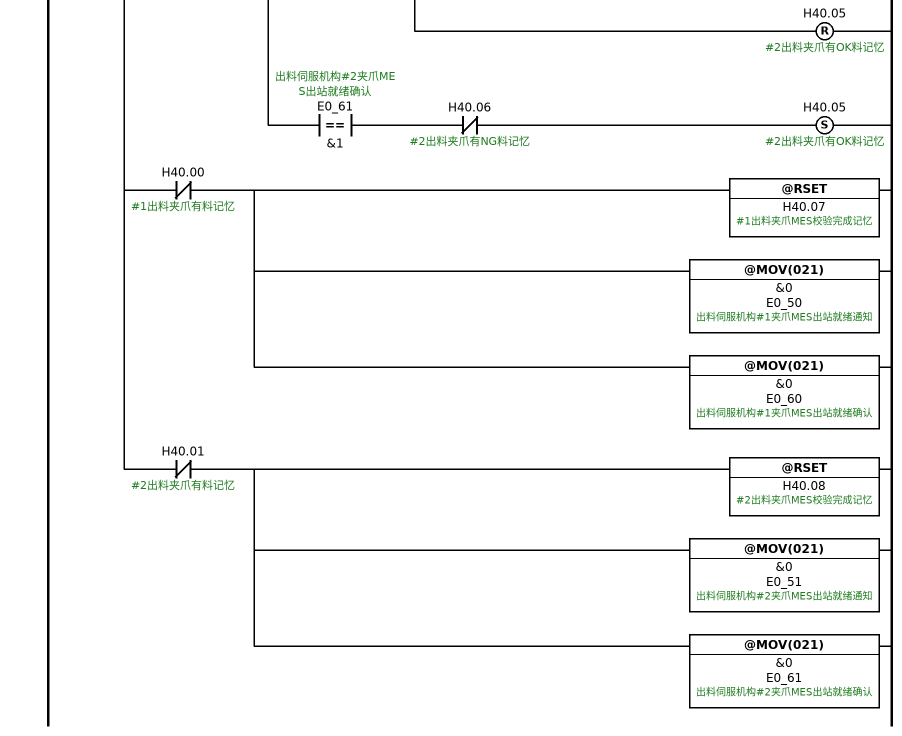
; [picture p408: 出料伺服机构 / Main, rungs 47-47]
; rung 47: 出料伺服机构MES出站校验完成记忆
LD P_On
OUT TR0
AND D1156.05  ; 下料模组夹爪夹紧
OUT TR1
ANDNOT H40.07  ; #1出料夹爪MES校验完成记忆
LD H40.00  ; #1出料夹爪有料记忆
LD>=(325) E0_60 &1  ; 出料伺服机构#1夹爪MES出站就绪确认  // #1出站就绪确认=0：未确认，1：确认OK，
OR H5.07  ; 电脑屏蔽-HMI
OR H5.10  ; 空跑程序
ANDLD
LDNOT H40.00  ; #1出料夹爪有料记忆  // 正常|清尾料时单料状况
AND H40.01  ; #2出料夹爪有料记忆
ORLD
ANDLD
@SET H40.07  ; #1出料夹爪MES校验完成记忆
LD TR1
ANDNOT H40.08  ; #2出料夹爪MES校验完成记忆
LD H40.01  ; #2出料夹爪有料记忆
LD>=(325) E0_61 &1  ; 出料伺服机构#2夹爪MES出站就绪确认  // #2出站就绪确认=0：未确认，1：确认OK，
OR H5.07  ; 电脑屏蔽-HMI
OR H5.10  ; 空跑程序
ANDLD
LDNOT H40.01  ; #2出料夹爪有料记忆  // 正常|清尾料时单料状况
AND H40.00  ; #1出料夹爪有料记忆
ORLD
ANDLD
@SET H40.08  ; #2出料夹爪MES校验完成记忆
LD TR0
AND H40.07  ; #1出料夹爪MES校验完成记忆
LDNOT H6.06  ; MES出站校验使用(1使用)
LD H6.06  ; MES出站校验使用(1使用)
OR P_On
LD H40.03  ; #1出料夹爪有OK料记忆
OR H40.04  ; #1出料夹爪有NG料记忆
ANDLD
ORLD
ANDLD
@MOV(021) &0 E0_50  ; 出料伺服机构#1夹爪MES出站就绪通知
LD TR0
AND H40.08  ; #2出料夹爪MES校验完成记忆
LDNOT H6.06  ; MES出站校验使用(1使用)
LD H6.06  ; MES出站校验使用(1使用)
OR P_On
LD H40.05  ; #2出料夹爪有OK料记忆
OR H40.06  ; #2出料夹爪有NG料记忆
ANDLD
ORLD
ANDLD
@MOV(021) &0 E0_51  ; 出料伺服机构#2夹爪MES出站就绪通知
LD TR0
LD H6.06  ; MES出站校验使用(1使用)
OR P_On
ANDLD
OUT TR1
AND>(320) E0_60 &1  ; 出料伺服机构#1夹爪MES出站就绪确认  // #1出站就绪确认=0：未确认，1：确认OK，
SET H40.04  ; #1出料夹爪有NG料记忆
RSET H40.03  ; #1出料夹爪有OK料记忆
LD TR1
AND=(300) E0_60 &1  ; 出料伺服机构#1夹爪MES出站就绪确认  // #1出站就绪确认=0：未确认，1：确认OK，
ANDNOT H40.04  ; #1出料夹爪有NG料记忆
SET H40.03  ; #1出料夹爪有OK料记忆
LD TR1
AND>(320) E0_61 &1  ; 出料伺服机构#2夹爪MES出站就绪确认  // #1出站就绪确认=0：未确认，1：确认OK，
SET H40.06  ; #2出料夹爪有NG料记忆
RSET H40.05  ; #2出料夹爪有OK料记忆
LD TR1
AND=(300) E0_61 &1  ; 出料伺服机构#2夹爪MES出站就绪确认  // #1出站就绪确认=0：未确认，1：确认OK，
ANDNOT H40.06  ; #2出料夹爪有NG料记忆
SET H40.05  ; #2出料夹爪有OK料记忆
LD TR0
ANDNOT H40.00  ; #1出料夹爪有料记忆
@RSET H40.07  ; #1出料夹爪MES校验完成记忆
@MOV(021) &0 E0_50  ; 出料伺服机构#1夹爪MES出站就绪通知
@MOV(021) &0 E0_60  ; 出料伺服机构#1夹爪MES出站就绪确认
LD TR0
ANDNOT H40.01  ; #2出料夹爪有料记忆
@RSET H40.08  ; #2出料夹爪MES校验完成记忆
@MOV(021) &0 E0_51  ; 出料伺服机构#2夹爪MES出站就绪通知
@MOV(021) &0 E0_61  ; 出料伺服机构#2夹爪MES出站就绪确认

### Section 出料伺服手动

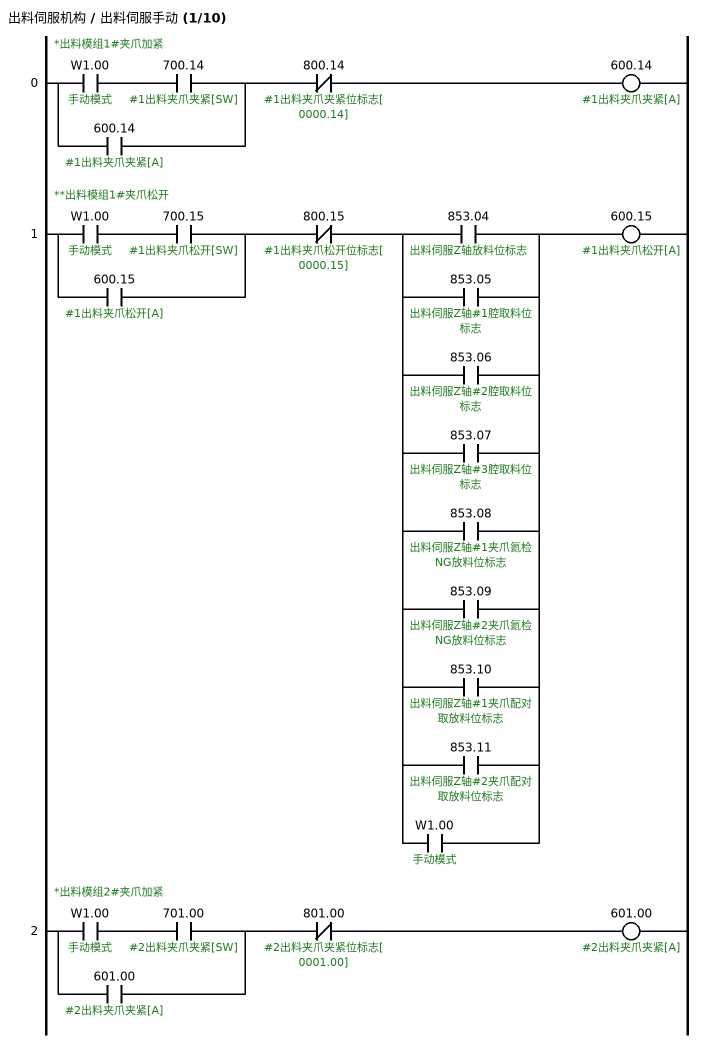
; rung 0: *出料模组1#夹爪加紧
LD W1.00  ; 手动模式
AND 700.14  ; #1出料夹爪夹紧[SW]
OR 600.14  ; #1出料夹爪夹紧[A]
ANDNOT 800.14  ; #1出料夹爪夹紧位标志[0000.14]
OUT 600.14  ; #1出料夹爪夹紧[A]
; rung 1: **出料模组1#夹爪松开
LD W1.00  ; 手动模式
AND 700.15  ; #1出料夹爪松开[SW]
OR 600.15  ; #1出料夹爪松开[A]
ANDNOT 800.15  ; #1出料夹爪松开位标志[0000.15]
LD 853.04  ; 出料伺服Z轴放料位标志
OR 853.05  ; 出料伺服Z轴#1腔取料位标志
OR 853.06  ; 出料伺服Z轴#2腔取料位标志
OR 853.07  ; 出料伺服Z轴#3腔取料位标志
OR 853.08  ; 出料伺服Z轴#1夹爪氦检NG放料位标志
OR 853.09  ; 出料伺服Z轴#2夹爪氦检NG放料位标志
OR 853.10  ; 出料伺服Z轴#1夹爪配对取放料位标志
OR 853.11  ; 出料伺服Z轴#2夹爪配对取放料位标志
OR W1.00  ; 手动模式
ANDLD
OUT 600.15  ; #1出料夹爪松开[A]
; rung 2: *出料模组2#夹爪加紧
LD W1.00  ; 手动模式
AND 701.00  ; #2出料夹爪夹紧[SW]
OR 601.00  ; #2出料夹爪夹紧[A]
ANDNOT 801.00  ; #2出料夹爪夹紧位标志[0001.00]
OUT 601.00  ; #2出料夹爪夹紧[A]

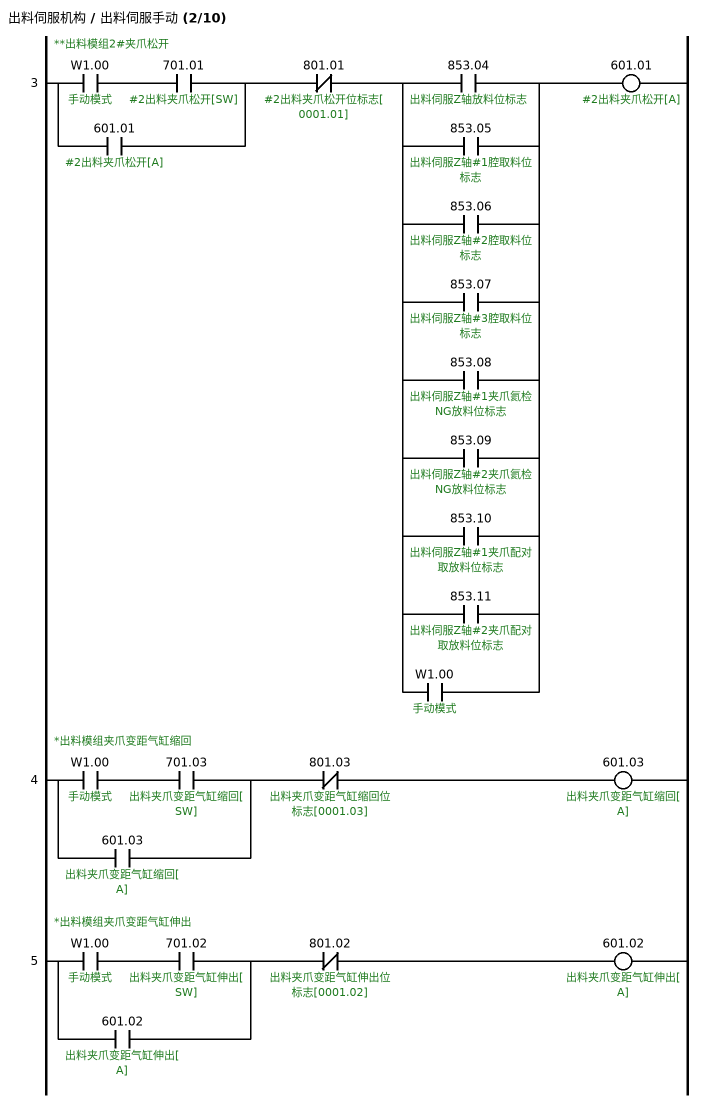
; rung 3: **出料模组2#夹爪松开
LD W1.00  ; 手动模式
AND 701.01  ; #2出料夹爪松开[SW]
OR 601.01  ; #2出料夹爪松开[A]
ANDNOT 801.01  ; #2出料夹爪松开位标志[0001.01]
LD 853.04  ; 出料伺服Z轴放料位标志
OR 853.05  ; 出料伺服Z轴#1腔取料位标志
OR 853.06  ; 出料伺服Z轴#2腔取料位标志
OR 853.07  ; 出料伺服Z轴#3腔取料位标志
OR 853.08  ; 出料伺服Z轴#1夹爪氦检NG放料位标志
OR 853.09  ; 出料伺服Z轴#2夹爪氦检NG放料位标志
OR 853.10  ; 出料伺服Z轴#1夹爪配对取放料位标志
OR 853.11  ; 出料伺服Z轴#2夹爪配对取放料位标志
OR W1.00  ; 手动模式
ANDLD
OUT 601.01  ; #2出料夹爪松开[A]
; rung 4: *出料模组夹爪变距气缸缩回
LD W1.00  ; 手动模式
AND 701.03  ; 出料夹爪变距气缸缩回[SW]
OR 601.03  ; 出料夹爪变距气缸缩回[A]
ANDNOT 801.03  ; 出料夹爪变距气缸缩回位标志[0001.03]
OUT 601.03  ; 出料夹爪变距气缸缩回[A]
; rung 5: *出料模组夹爪变距气缸伸出
LD W1.00  ; 手动模式
AND 701.02  ; 出料夹爪变距气缸伸出[SW]
OR 601.02  ; 出料夹爪变距气缸伸出[A]
ANDNOT 801.02  ; 出料夹爪变距气缸伸出位标志[0001.02]
OUT 601.02  ; 出料夹爪变距气缸伸出[A]

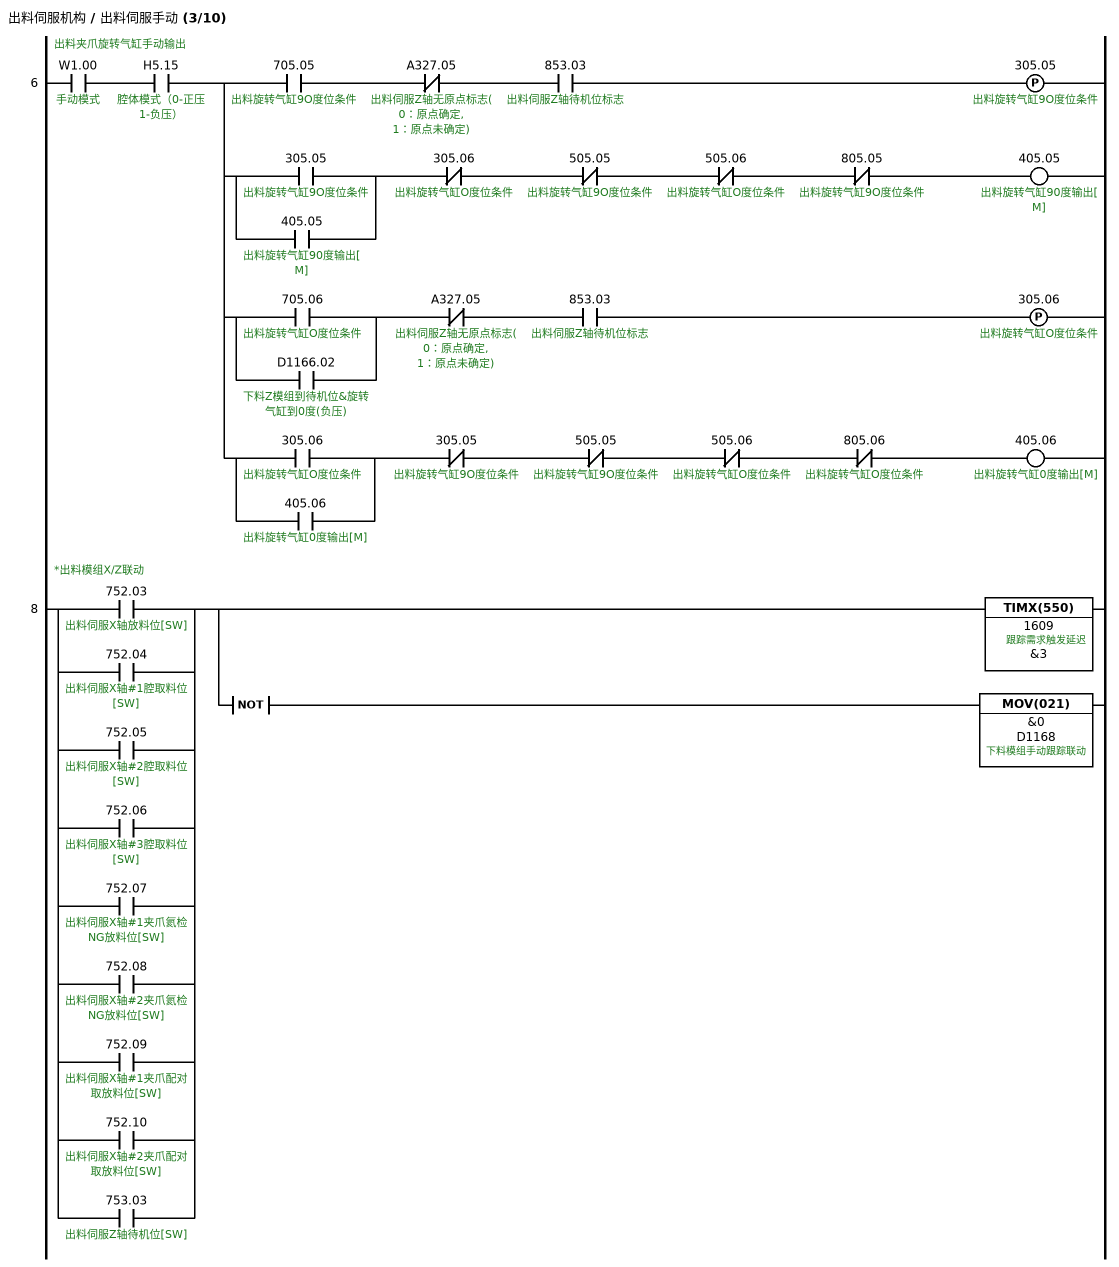
; rung 6: 出料夹爪旋转气缸手动输出
LD W1.00  ; 手动模式
AND H5.15  ; 腔体模式（0-正压 1-负压）
OUT TR0
AND 705.05  ; 出料旋转气缸9O度位条件
ANDNOT A327.05  ; 出料伺服Z轴无原点标志(0：原点确定,1：原点未确定)
AND 853.03  ; 出料伺服Z轴待机位标志
DIFU(013) 305.05  ; 出料旋转气缸9O度位条件
LD TR0
LD 305.05  ; 出料旋转气缸9O度位条件
OR 405.05  ; 出料旋转气缸90度输出[M]
ANDLD
ANDNOT 305.06  ; 出料旋转气缸O度位条件
ANDNOT 505.05  ; 出料旋转气缸9O度位条件
ANDNOT 505.06  ; 出料旋转气缸O度位条件
ANDNOT 805.05  ; 出料旋转气缸9O度位条件
OUT 405.05  ; 出料旋转气缸90度输出[M]
LD TR0
LD 705.06  ; 出料旋转气缸O度位条件
OR D1166.02  ; 下料Z模组到待机位&旋转气缸到0度(负压)
ANDLD
ANDNOT A327.05  ; 出料伺服Z轴无原点标志(0：原点确定,1：原点未确定)
AND 853.03  ; 出料伺服Z轴待机位标志
DIFU(013) 305.06  ; 出料旋转气缸O度位条件
LD TR0
LD 305.06  ; 出料旋转气缸O度位条件
OR 405.06  ; 出料旋转气缸0度输出[M]
ANDLD
ANDNOT 305.05  ; 出料旋转气缸9O度位条件
ANDNOT 505.05  ; 出料旋转气缸9O度位条件
ANDNOT 505.06  ; 出料旋转气缸O度位条件
ANDNOT 805.06  ; 出料旋转气缸O度位条件
OUT 405.06  ; 出料旋转气缸0度输出[M]
; rung 7: ************************** / **************************
; rung 8: *出料模组X/Z联动
LD 752.03  ; 出料伺服X轴放料位[SW]
OR 752.04  ; 出料伺服X轴#1腔取料位[SW]
OR 752.05  ; 出料伺服X轴#2腔取料位[SW]
OR 752.06  ; 出料伺服X轴#3腔取料位[SW]
OR 752.07  ; 出料伺服X轴#1夹爪氦检NG放料位[SW]
OR 752.08  ; 出料伺服X轴#2夹爪氦检NG放料位[SW]
OR 752.09  ; 出料伺服X轴#1夹爪配对取放料位[SW]
OR 752.10  ; 出料伺服X轴#2夹爪配对取放料位[SW]
OR 753.03  ; 出料伺服Z轴待机位[SW]
TIMX(550) 1609 &3  ; 跟踪需求触发延迟
NOT(520)
MOV(021) &0 D1168  ; 下料模组手动跟踪联动

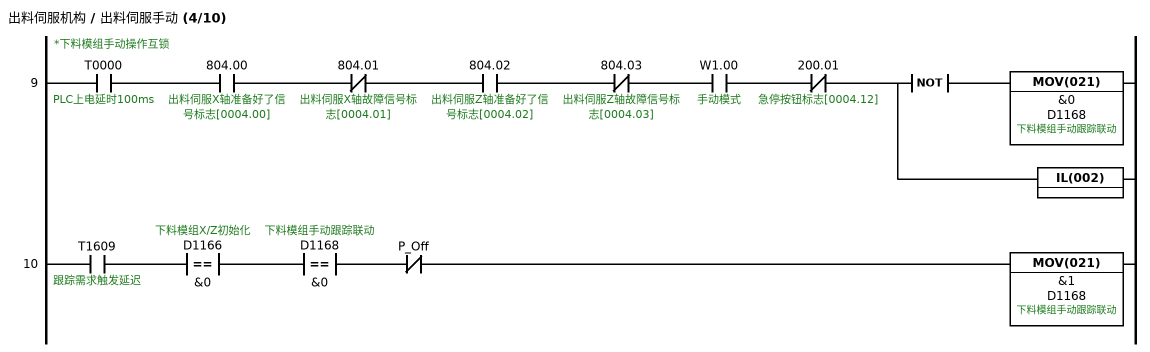
; rung 9: *下料模组手动操作互锁
LD T0000  ; PLC上电延时100ms
AND 804.00  ; 出料伺服X轴准备好了信号标志[0004.00]
ANDNOT 804.01  ; 出料伺服X轴故障信号标志[0004.01]
AND 804.02  ; 出料伺服Z轴准备好了信号标志[0004.02]
ANDNOT 804.03  ; 出料伺服Z轴故障信号标志[0004.03]
AND W1.00  ; 手动模式
ANDNOT 200.01  ; 急停按钮标志[0004.12]
OUT TR0
NOT(520)
MOV(021) &0 D1168  ; 下料模组手动跟踪联动
LD TR0
IL(002)
; rung 10
LD T1609  ; 跟踪需求触发延迟
AND=(300) D1166 &0  ; 下料模组X/Z初始化
AND=(300) D1168 &0  ; 下料模组手动跟踪联动
ANDNOT P_Off
MOV(021) &1 D1168  ; 下料模组手动跟踪联动

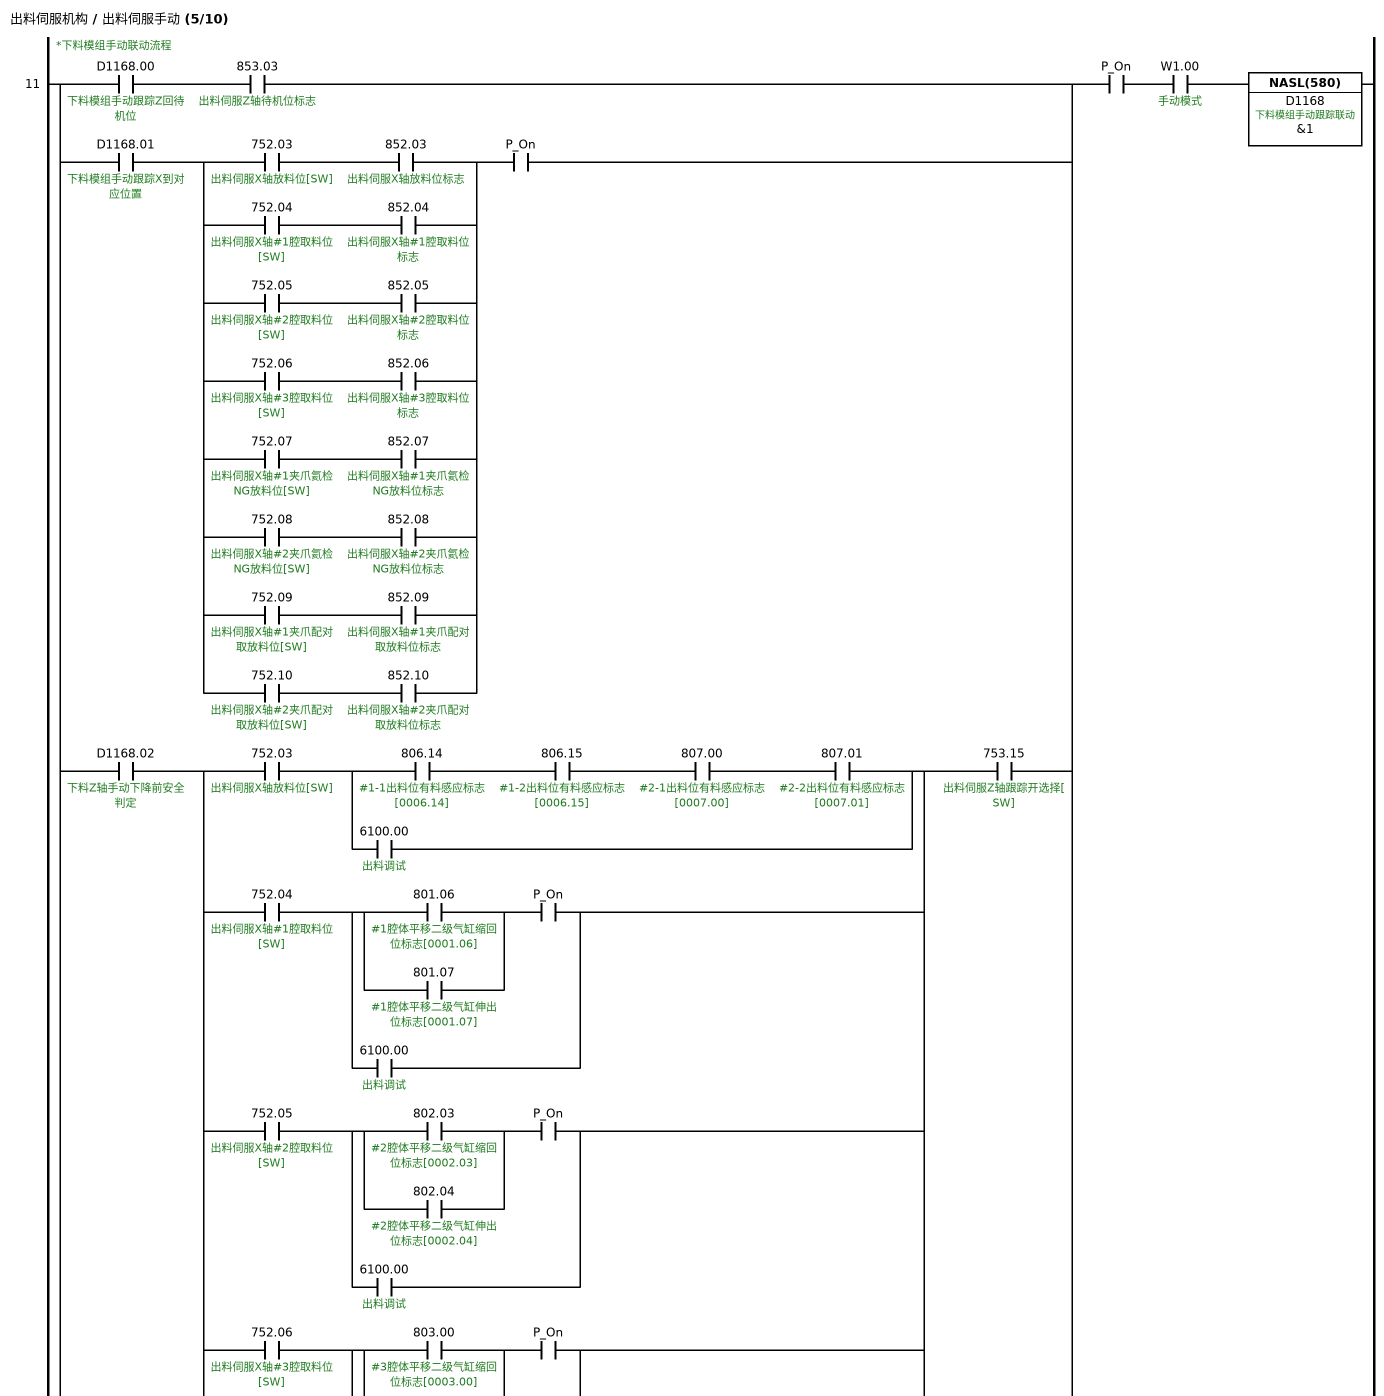

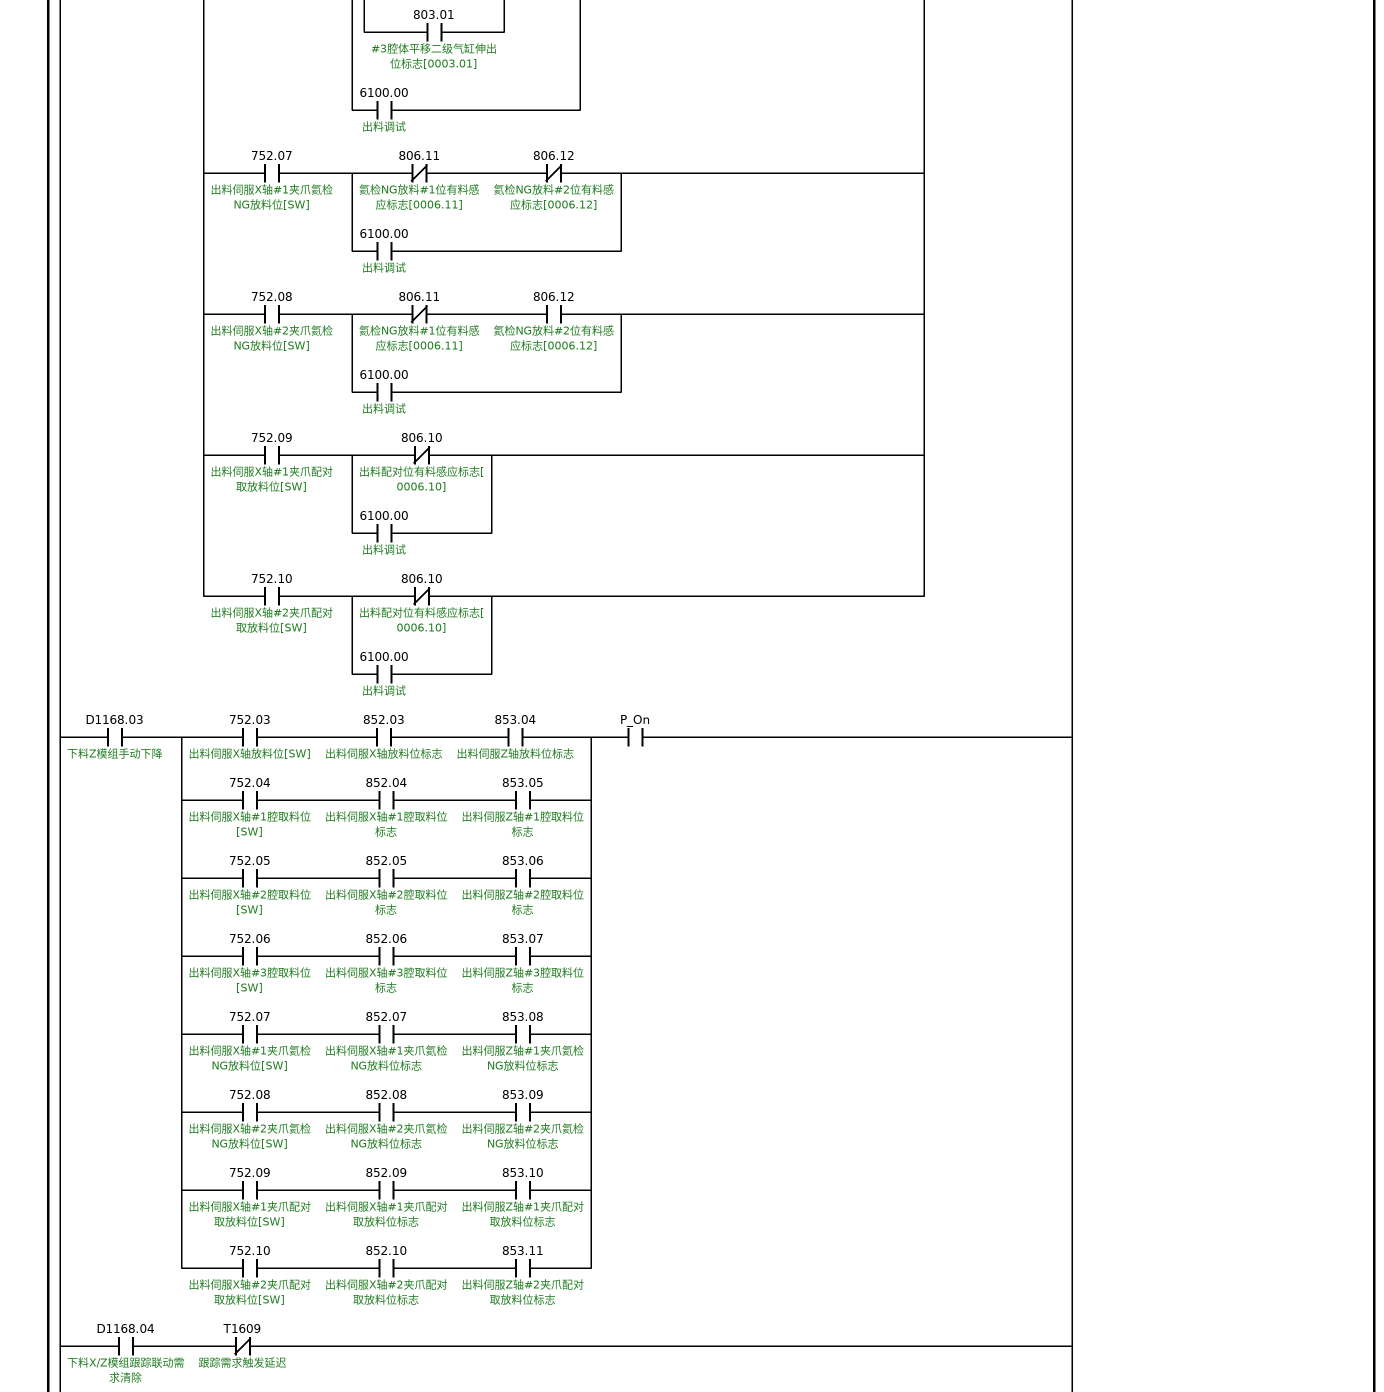

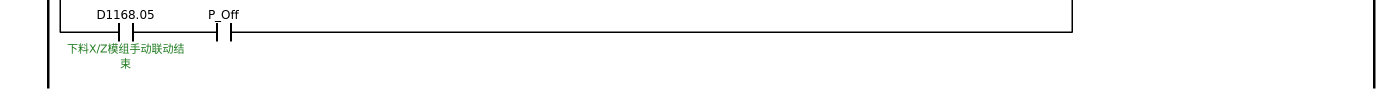
; rung 11: *下料模组手动联动流程
LD D1168.00  ; 下料模组手动跟踪Z回待机位
AND 853.03  ; 出料伺服Z轴待机位标志
LD D1168.01  ; 下料模组手动跟踪X到对应位置
LD 752.03  ; 出料伺服X轴放料位[SW]
AND 852.03  ; 出料伺服X轴放料位标志
LD 752.04  ; 出料伺服X轴#1腔取料位[SW]
AND 852.04  ; 出料伺服X轴#1腔取料位标志
ORLD
LD 752.05  ; 出料伺服X轴#2腔取料位[SW]
AND 852.05  ; 出料伺服X轴#2腔取料位标志
ORLD
LD 752.06  ; 出料伺服X轴#3腔取料位[SW]
AND 852.06  ; 出料伺服X轴#3腔取料位标志
ORLD
LD 752.07  ; 出料伺服X轴#1夹爪氦检NG放料位[SW]
AND 852.07  ; 出料伺服X轴#1夹爪氦检NG放料位标志
ORLD
LD 752.08  ; 出料伺服X轴#2夹爪氦检NG放料位[SW]
AND 852.08  ; 出料伺服X轴#2夹爪氦检NG放料位标志
ORLD
LD 752.09  ; 出料伺服X轴#1夹爪配对取放料位[SW]
AND 852.09  ; 出料伺服X轴#1夹爪配对取放料位标志
ORLD
LD 752.10  ; 出料伺服X轴#2夹爪配对取放料位[SW]
AND 852.10  ; 出料伺服X轴#2夹爪配对取放料位标志
ORLD
ANDLD
AND P_On
ORLD
LD D1168.02  ; 下料Z轴手动下降前安全判定
LD 752.03  ; 出料伺服X轴放料位[SW]
LD 806.14  ; #1-1出料位有料感应标志[0006.14]
AND 806.15  ; #1-2出料位有料感应标志[0006.15]
AND 807.00  ; #2-1出料位有料感应标志[0007.00]
AND 807.01  ; #2-2出料位有料感应标志[0007.01]
OR 6100.00  ; 出料调试
ANDLD
LD 752.04  ; 出料伺服X轴#1腔取料位[SW]
LD 801.06  ; #1腔体平移二级气缸缩回位标志[0001.06]
OR 801.07  ; #1腔体平移二级气缸伸出位标志[0001.07]
AND P_On
OR 6100.00  ; 出料调试
ANDLD
ORLD
LD 752.05  ; 出料伺服X轴#2腔取料位[SW]
LD 802.03  ; #2腔体平移二级气缸缩回位标志[0002.03]
OR 802.04  ; #2腔体平移二级气缸伸出位标志[0002.04]
AND P_On
OR 6100.00  ; 出料调试
ANDLD
ORLD
LD 752.06  ; 出料伺服X轴#3腔取料位[SW]
LD 803.00  ; #3腔体平移二级气缸缩回位标志[0003.00]
OR 803.01  ; #3腔体平移二级气缸伸出位标志[0003.01]
AND P_On
OR 6100.00  ; 出料调试
ANDLD
ORLD
LD 752.07  ; 出料伺服X轴#1夹爪氦检NG放料位[SW]
LDNOT 806.11  ; 氦检NG放料#1位有料感应标志[0006.11]
ANDNOT 806.12  ; 氦检NG放料#2位有料感应标志[0006.12]
OR 6100.00  ; 出料调试
ANDLD
ORLD
LD 752.08  ; 出料伺服X轴#2夹爪氦检NG放料位[SW]
LDNOT 806.11  ; 氦检NG放料#1位有料感应标志[0006.11]
AND 806.12  ; 氦检NG放料#2位有料感应标志[0006.12]
OR 6100.00  ; 出料调试
ANDLD
ORLD
LD 752.09  ; 出料伺服X轴#1夹爪配对取放料位[SW]
LDNOT 806.10  ; 出料配对位有料感应标志[0006.10]
OR 6100.00  ; 出料调试
ANDLD
ORLD
LD 752.10  ; 出料伺服X轴#2夹爪配对取放料位[SW]
LDNOT 806.10  ; 出料配对位有料感应标志[0006.10]
OR 6100.00  ; 出料调试
ANDLD
ORLD
ANDLD
AND 753.15  ; 出料伺服Z轴跟踪开选择[SW]
ORLD
LD D1168.03  ; 下料Z模组手动下降
LD 752.03  ; 出料伺服X轴放料位[SW]
AND 852.03  ; 出料伺服X轴放料位标志
AND 853.04  ; 出料伺服Z轴放料位标志
LD 752.04  ; 出料伺服X轴#1腔取料位[SW]
AND 852.04  ; 出料伺服X轴#1腔取料位标志
AND 853.05  ; 出料伺服Z轴#1腔取料位标志
ORLD
LD 752.05  ; 出料伺服X轴#2腔取料位[SW]
AND 852.05  ; 出料伺服X轴#2腔取料位标志
AND 853.06  ; 出料伺服Z轴#2腔取料位标志
ORLD
LD 752.06  ; 出料伺服X轴#3腔取料位[SW]
AND 852.06  ; 出料伺服X轴#3腔取料位标志
AND 853.07  ; 出料伺服Z轴#3腔取料位标志
ORLD
LD 752.07  ; 出料伺服X轴#1夹爪氦检NG放料位[SW]
AND 852.07  ; 出料伺服X轴#1夹爪氦检NG放料位标志
AND 853.08  ; 出料伺服Z轴#1夹爪氦检NG放料位标志
ORLD
LD 752.08  ; 出料伺服X轴#2夹爪氦检NG放料位[SW]
AND 852.08  ; 出料伺服X轴#2夹爪氦检NG放料位标志
AND 853.09  ; 出料伺服Z轴#2夹爪氦检NG放料位标志
ORLD
LD 752.09  ; 出料伺服X轴#1夹爪配对取放料位[SW]
AND 852.09  ; 出料伺服X轴#1夹爪配对取放料位标志
AND 853.10  ; 出料伺服Z轴#1夹爪配对取放料位标志
ORLD
LD 752.10  ; 出料伺服X轴#2夹爪配对取放料位[SW]
AND 852.10  ; 出料伺服X轴#2夹爪配对取放料位标志
AND 853.11  ; 出料伺服Z轴#2夹爪配对取放料位标志
ORLD
ANDLD
AND P_On
ORLD
LD D1168.04  ; 下料X/Z模组跟踪联动需求清除
ANDNOT T1609  ; 跟踪需求触发延迟
ORLD
LD D1168.05  ; 下料X/Z模组手动联动结束
AND P_Off
ORLD
AND P_On
AND W1.00  ; 手动模式
NASL(580) D1168 &1  ; 下料模组手动跟踪联动

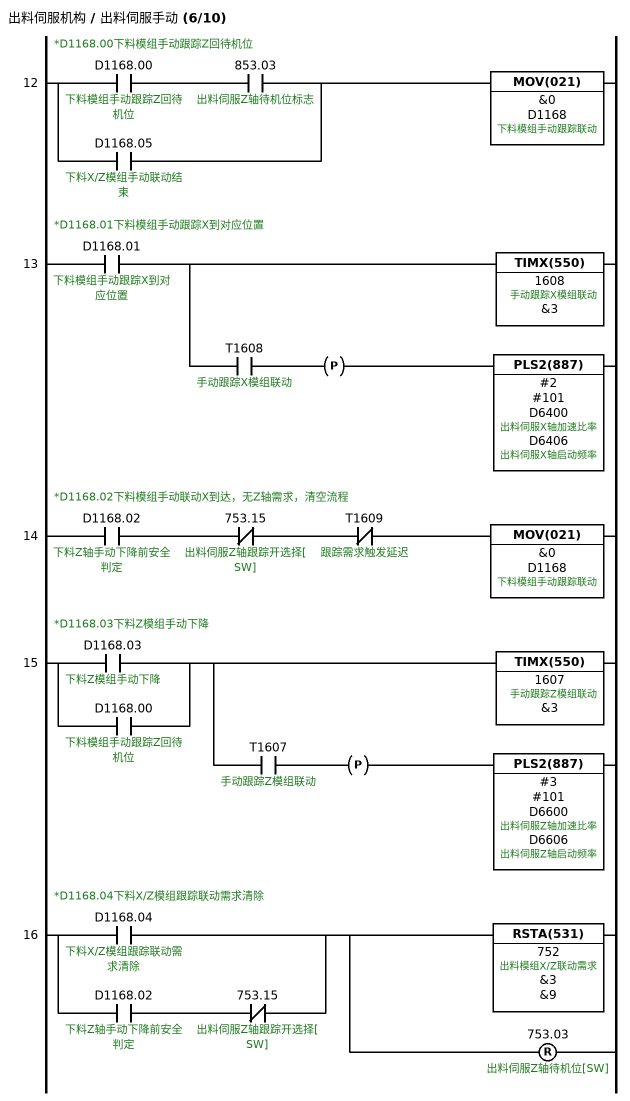
; rung 12: *D1168.00下料模组手动跟踪Z回待机位
LD D1168.00  ; 下料模组手动跟踪Z回待机位
AND 853.03  ; 出料伺服Z轴待机位标志
OR D1168.05  ; 下料X/Z模组手动联动结束
MOV(021) &0 D1168  ; 下料模组手动跟踪联动
; rung 13: *D1168.01下料模组手动跟踪X到对应位置
LD D1168.01  ; 下料模组手动跟踪X到对应位置
TIMX(550) 1608 &3  ; 手动跟踪X模组联动
AND T1608  ; 手动跟踪X模组联动
UP(521)
PLS2(887) #2 #101 D6400 D6406  ; 出料伺服X轴加速比率, 出料伺服X轴启动频率
; rung 14: *D1168.02下料模组手动联动X到达，无Z轴需求，清空流程
LD D1168.02  ; 下料Z轴手动下降前安全判定
ANDNOT 753.15  ; 出料伺服Z轴跟踪开选择[SW]
ANDNOT T1609  ; 跟踪需求触发延迟
MOV(021) &0 D1168  ; 下料模组手动跟踪联动
; rung 15: *D1168.03下料Z模组手动下降
LD D1168.03  ; 下料Z模组手动下降
OR D1168.00  ; 下料模组手动跟踪Z回待机位
TIMX(550) 1607 &3  ; 手动跟踪Z模组联动
AND T1607  ; 手动跟踪Z模组联动
UP(521)
PLS2(887) #3 #101 D6600 D6606  ; 出料伺服Z轴加速比率, 出料伺服Z轴启动频率
; rung 16: *D1168.04下料X/Z模组跟踪联动需求清除
LD D1168.04  ; 下料X/Z模组跟踪联动需求清除
LD D1168.02  ; 下料Z轴手动下降前安全判定
ANDNOT 753.15  ; 出料伺服Z轴跟踪开选择[SW]
ORLD
RSTA(531) 752 &3 &9  ; 出料模组X/Z联动需求
RSET 753.03  ; 出料伺服Z轴待机位[SW]

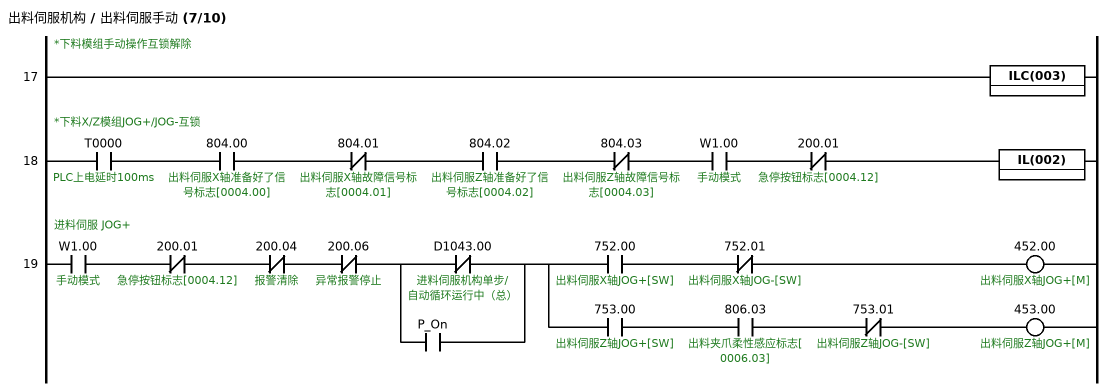
; rung 17: *下料模组手动操作互锁解除
ILC(003)
; rung 18: *下料X/Z模组JOG+/JOG-互锁
LD T0000  ; PLC上电延时100ms
AND 804.00  ; 出料伺服X轴准备好了信号标志[0004.00]
ANDNOT 804.01  ; 出料伺服X轴故障信号标志[0004.01]
AND 804.02  ; 出料伺服Z轴准备好了信号标志[0004.02]
ANDNOT 804.03  ; 出料伺服Z轴故障信号标志[0004.03]
AND W1.00  ; 手动模式
ANDNOT 200.01  ; 急停按钮标志[0004.12]
IL(002)
; rung 19: 进料伺服 JOG+
LD W1.00  ; 手动模式
ANDNOT 200.01  ; 急停按钮标志[0004.12]
ANDNOT 200.04  ; 报警清除
ANDNOT 200.06  ; 异常报警停止
LDNOT D1043.00  ; 进料伺服机构单步/自动循环运行中（总）
OR P_On
ANDLD
OUT TR0
AND 752.00  ; 出料伺服X轴JOG+[SW]
ANDNOT 752.01  ; 出料伺服X轴JOG-[SW]
OUT 452.00  ; 出料伺服X轴JOG+[M]
LD TR0
AND 753.00  ; 出料伺服Z轴JOG+[SW]
AND 806.03  ; 出料夹爪柔性感应标志[0006.03]
ANDNOT 753.01  ; 出料伺服Z轴JOG-[SW]
OUT 453.00  ; 出料伺服Z轴JOG+[M]

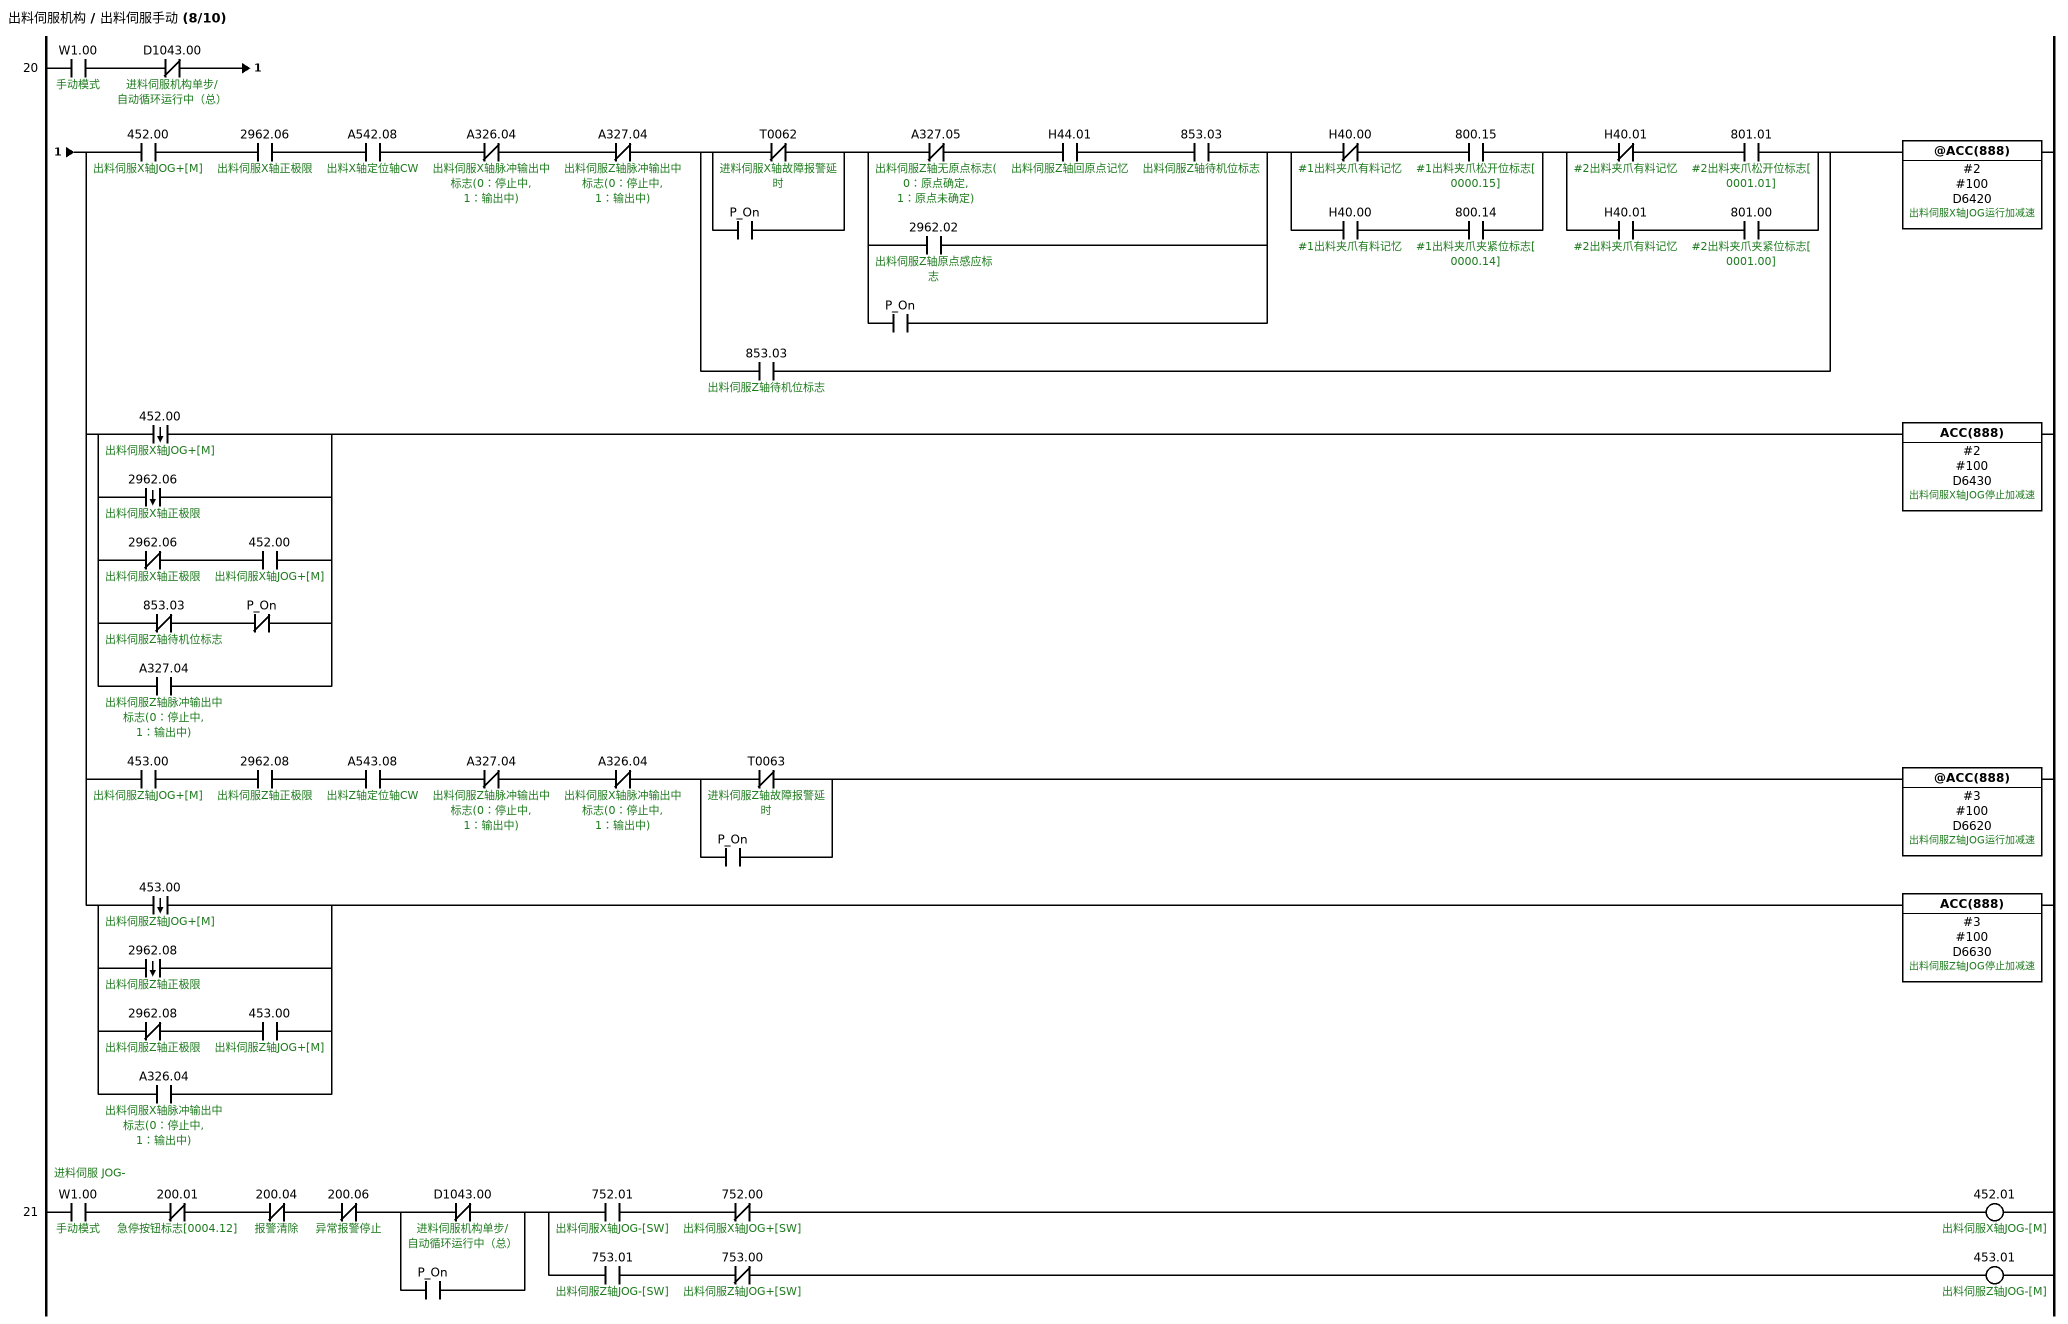
; rung 20
LD W1.00  ; 手动模式
ANDNOT D1043.00  ; 进料伺服机构单步/自动循环运行中（总）
OUT TR0
AND 452.00  ; 出料伺服X轴JOG+[M]
AND 2962.06  ; 出料伺服X轴正极限
AND A542.08  ; 出料X轴定位轴CW
ANDNOT A326.04  ; 出料伺服X轴脉冲输出中标志(0：停止中,1：输出中)
ANDNOT A327.04  ; 出料伺服Z轴脉冲输出中标志(0：停止中,1：输出中)
LDNOT T0062  ; 进料伺服X轴故障报警延时
OR P_On
LDNOT A327.05  ; 出料伺服Z轴无原点标志(0：原点确定,1：原点未确定)
AND H44.01  ; 出料伺服Z轴回原点记忆
AND 853.03  ; 出料伺服Z轴待机位标志
OR 2962.02  ; 出料伺服Z轴原点感应标志
OR P_On
ANDLD
LDNOT H40.00  ; #1出料夹爪有料记忆
AND 800.15  ; #1出料夹爪松开位标志[0000.15]
LD H40.00  ; #1出料夹爪有料记忆
AND 800.14  ; #1出料夹爪夹紧位标志[0000.14]
ORLD
ANDLD
LDNOT H40.01  ; #2出料夹爪有料记忆
AND 801.01  ; #2出料夹爪松开位标志[0001.01]
LD H40.01  ; #2出料夹爪有料记忆
AND 801.00  ; #2出料夹爪夹紧位标志[0001.00]
ORLD
ANDLD
OR 853.03  ; 出料伺服Z轴待机位标志
ANDLD
@ACC(888) #2 #100 D6420  ; 出料伺服X轴JOG运行加减速
LD TR0
%LD 452.00  ; 出料伺服X轴JOG+[M]
%OR 2962.06  ; 出料伺服X轴正极限
LDNOT 2962.06  ; 出料伺服X轴正极限
AND 452.00  ; 出料伺服X轴JOG+[M]
ORLD
LDNOT 853.03  ; 出料伺服Z轴待机位标志
ANDNOT P_On
ORLD
OR A327.04  ; 出料伺服Z轴脉冲输出中标志(0：停止中,1：输出中)
ANDLD
ACC(888) #2 #100 D6430  ; 出料伺服X轴JOG停止加减速
LD TR0
AND 453.00  ; 出料伺服Z轴JOG+[M]
AND 2962.08  ; 出料伺服Z轴正极限
AND A543.08  ; 出料Z轴定位轴CW
ANDNOT A327.04  ; 出料伺服Z轴脉冲输出中标志(0：停止中,1：输出中)
ANDNOT A326.04  ; 出料伺服X轴脉冲输出中标志(0：停止中,1：输出中)
LDNOT T0063  ; 进料伺服Z轴故障报警延时
OR P_On
ANDLD
@ACC(888) #3 #100 D6620  ; 出料伺服Z轴JOG运行加减速
LD TR0
%LD 453.00  ; 出料伺服Z轴JOG+[M]
%OR 2962.08  ; 出料伺服Z轴正极限
LDNOT 2962.08  ; 出料伺服Z轴正极限
AND 453.00  ; 出料伺服Z轴JOG+[M]
ORLD
OR A326.04  ; 出料伺服X轴脉冲输出中标志(0：停止中,1：输出中)
ANDLD
ACC(888) #3 #100 D6630  ; 出料伺服Z轴JOG停止加减速
; rung 21: 进料伺服 JOG-
LD W1.00  ; 手动模式
ANDNOT 200.01  ; 急停按钮标志[0004.12]
ANDNOT 200.04  ; 报警清除
ANDNOT 200.06  ; 异常报警停止
LDNOT D1043.00  ; 进料伺服机构单步/自动循环运行中（总）
OR P_On
ANDLD
OUT TR0
AND 752.01  ; 出料伺服X轴JOG-[SW]
ANDNOT 752.00  ; 出料伺服X轴JOG+[SW]
OUT 452.01  ; 出料伺服X轴JOG-[M]
LD TR0
AND 753.01  ; 出料伺服Z轴JOG-[SW]
ANDNOT 753.00  ; 出料伺服Z轴JOG+[SW]
OUT 453.01  ; 出料伺服Z轴JOG-[M]

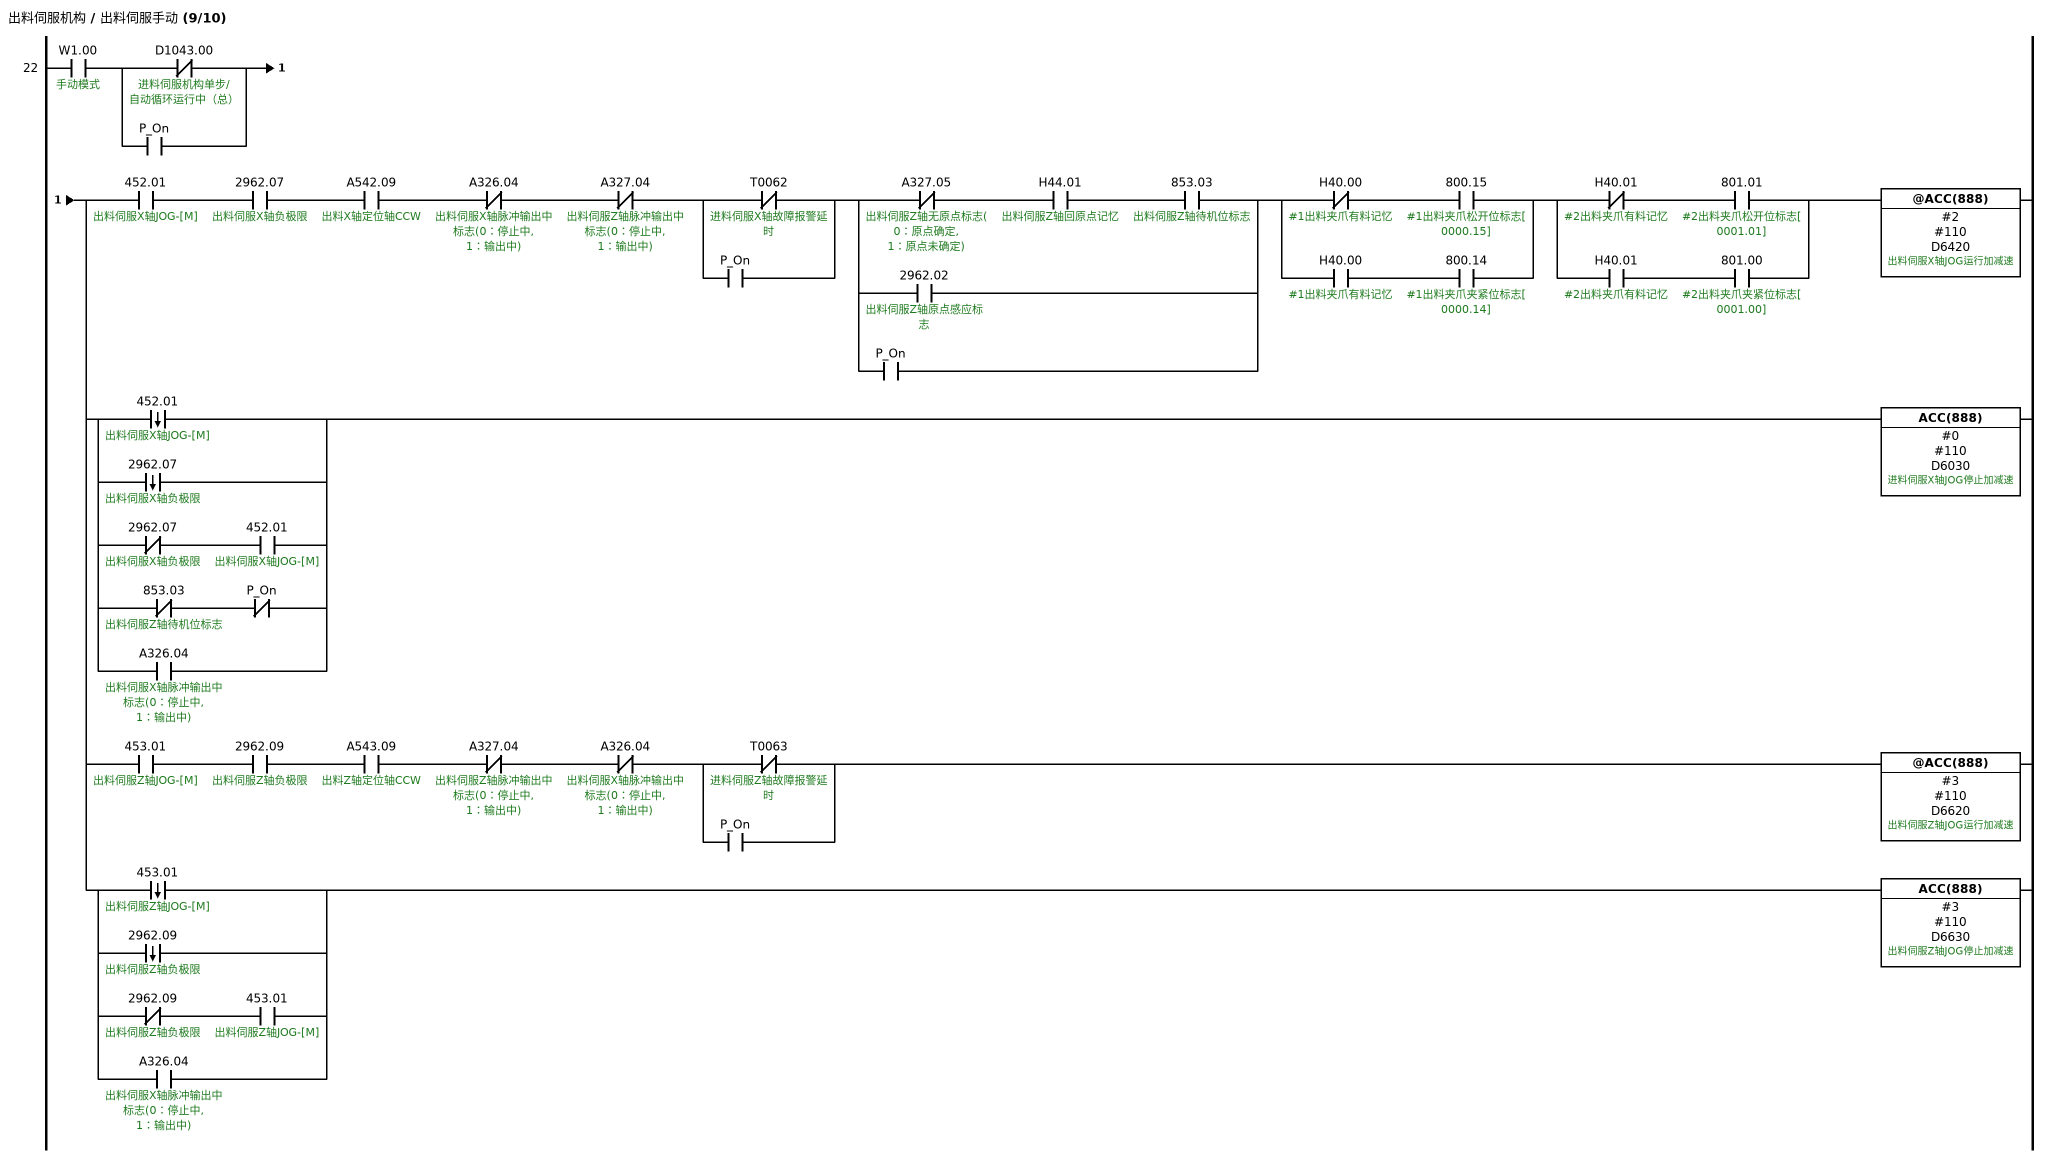
; rung 22
LD W1.00  ; 手动模式
LDNOT D1043.00  ; 进料伺服机构单步/自动循环运行中（总）
OR P_On
ANDLD
OUT TR0
AND 452.01  ; 出料伺服X轴JOG-[M]
AND 2962.07  ; 出料伺服X轴负极限
AND A542.09  ; 出料X轴定位轴CCW
ANDNOT A326.04  ; 出料伺服X轴脉冲输出中标志(0：停止中,1：输出中)
ANDNOT A327.04  ; 出料伺服Z轴脉冲输出中标志(0：停止中,1：输出中)
LDNOT T0062  ; 进料伺服X轴故障报警延时
OR P_On
ANDLD
LDNOT A327.05  ; 出料伺服Z轴无原点标志(0：原点确定,1：原点未确定)
AND H44.01  ; 出料伺服Z轴回原点记忆
AND 853.03  ; 出料伺服Z轴待机位标志
OR 2962.02  ; 出料伺服Z轴原点感应标志
OR P_On
ANDLD
LDNOT H40.00  ; #1出料夹爪有料记忆
AND 800.15  ; #1出料夹爪松开位标志[0000.15]
LD H40.00  ; #1出料夹爪有料记忆
AND 800.14  ; #1出料夹爪夹紧位标志[0000.14]
ORLD
ANDLD
LDNOT H40.01  ; #2出料夹爪有料记忆
AND 801.01  ; #2出料夹爪松开位标志[0001.01]
LD H40.01  ; #2出料夹爪有料记忆
AND 801.00  ; #2出料夹爪夹紧位标志[0001.00]
ORLD
ANDLD
@ACC(888) #2 #110 D6420  ; 出料伺服X轴JOG运行加减速
LD TR0
%LD 452.01  ; 出料伺服X轴JOG-[M]
%OR 2962.07  ; 出料伺服X轴负极限
LDNOT 2962.07  ; 出料伺服X轴负极限
AND 452.01  ; 出料伺服X轴JOG-[M]
ORLD
LDNOT 853.03  ; 出料伺服Z轴待机位标志
ANDNOT P_On
ORLD
OR A326.04  ; 出料伺服X轴脉冲输出中标志(0：停止中,1：输出中)
ANDLD
ACC(888) #0 #110 D6030  ; 进料伺服X轴JOG停止加减速
LD TR0
AND 453.01  ; 出料伺服Z轴JOG-[M]
AND 2962.09  ; 出料伺服Z轴负极限
AND A543.09  ; 出料Z轴定位轴CCW
ANDNOT A327.04  ; 出料伺服Z轴脉冲输出中标志(0：停止中,1：输出中)
ANDNOT A326.04  ; 出料伺服X轴脉冲输出中标志(0：停止中,1：输出中)
LDNOT T0063  ; 进料伺服Z轴故障报警延时
OR P_On
ANDLD
@ACC(888) #3 #110 D6620  ; 出料伺服Z轴JOG运行加减速
LD TR0
%LD 453.01  ; 出料伺服Z轴JOG-[M]
%OR 2962.09  ; 出料伺服Z轴负极限
LDNOT 2962.09  ; 出料伺服Z轴负极限
AND 453.01  ; 出料伺服Z轴JOG-[M]
ORLD
OR A326.04  ; 出料伺服X轴脉冲输出中标志(0：停止中,1：输出中)
ANDLD
ACC(888) #3 #110 D6630  ; 出料伺服Z轴JOG停止加减速

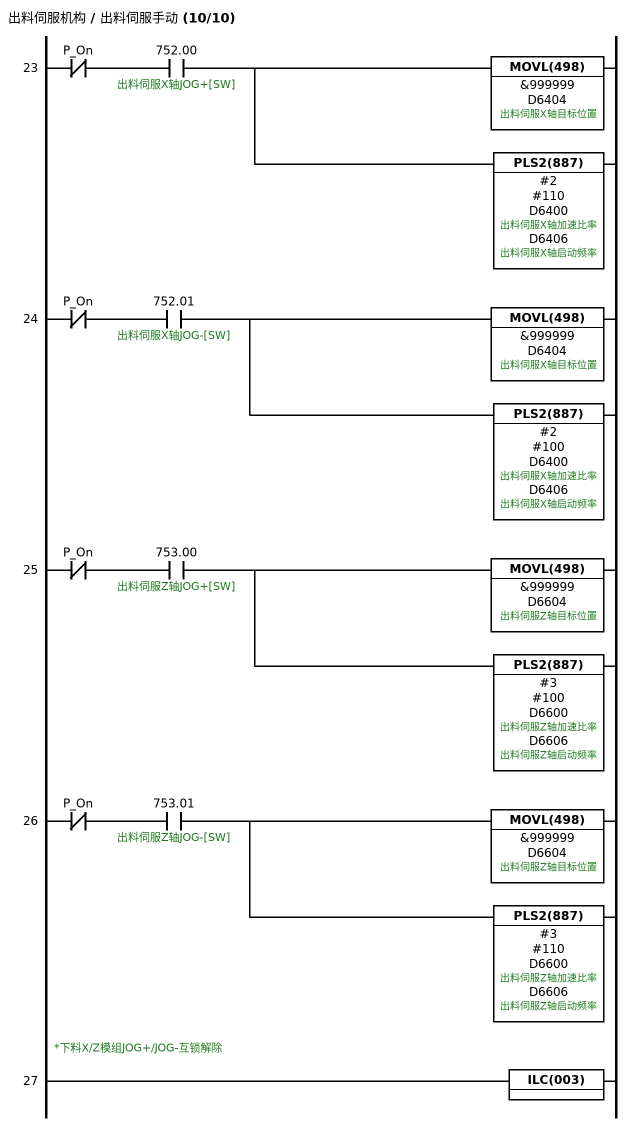
; rung 23
LDNOT P_On
AND 752.00  ; 出料伺服X轴JOG+[SW]
MOVL(498) &999999 D6404  ; 出料伺服X轴目标位置
PLS2(887) #2 #110 D6400 D6406  ; 出料伺服X轴加速比率, 出料伺服X轴启动频率
; rung 24
LDNOT P_On
AND 752.01  ; 出料伺服X轴JOG-[SW]
MOVL(498) &999999 D6404  ; 出料伺服X轴目标位置
PLS2(887) #2 #100 D6400 D6406  ; 出料伺服X轴加速比率, 出料伺服X轴启动频率
; rung 25
LDNOT P_On
AND 753.00  ; 出料伺服Z轴JOG+[SW]
MOVL(498) &999999 D6604  ; 出料伺服Z轴目标位置
PLS2(887) #3 #100 D6600 D6606  ; 出料伺服Z轴加速比率, 出料伺服Z轴启动频率
; rung 26
LDNOT P_On
AND 753.01  ; 出料伺服Z轴JOG-[SW]
MOVL(498) &999999 D6604  ; 出料伺服Z轴目标位置
PLS2(887) #3 #110 D6600 D6606  ; 出料伺服Z轴加速比率, 出料伺服Z轴启动频率
; rung 27: *下料X/Z模组JOG+/JOG-互锁解除
ILC(003)

### Section 出料伺服自动

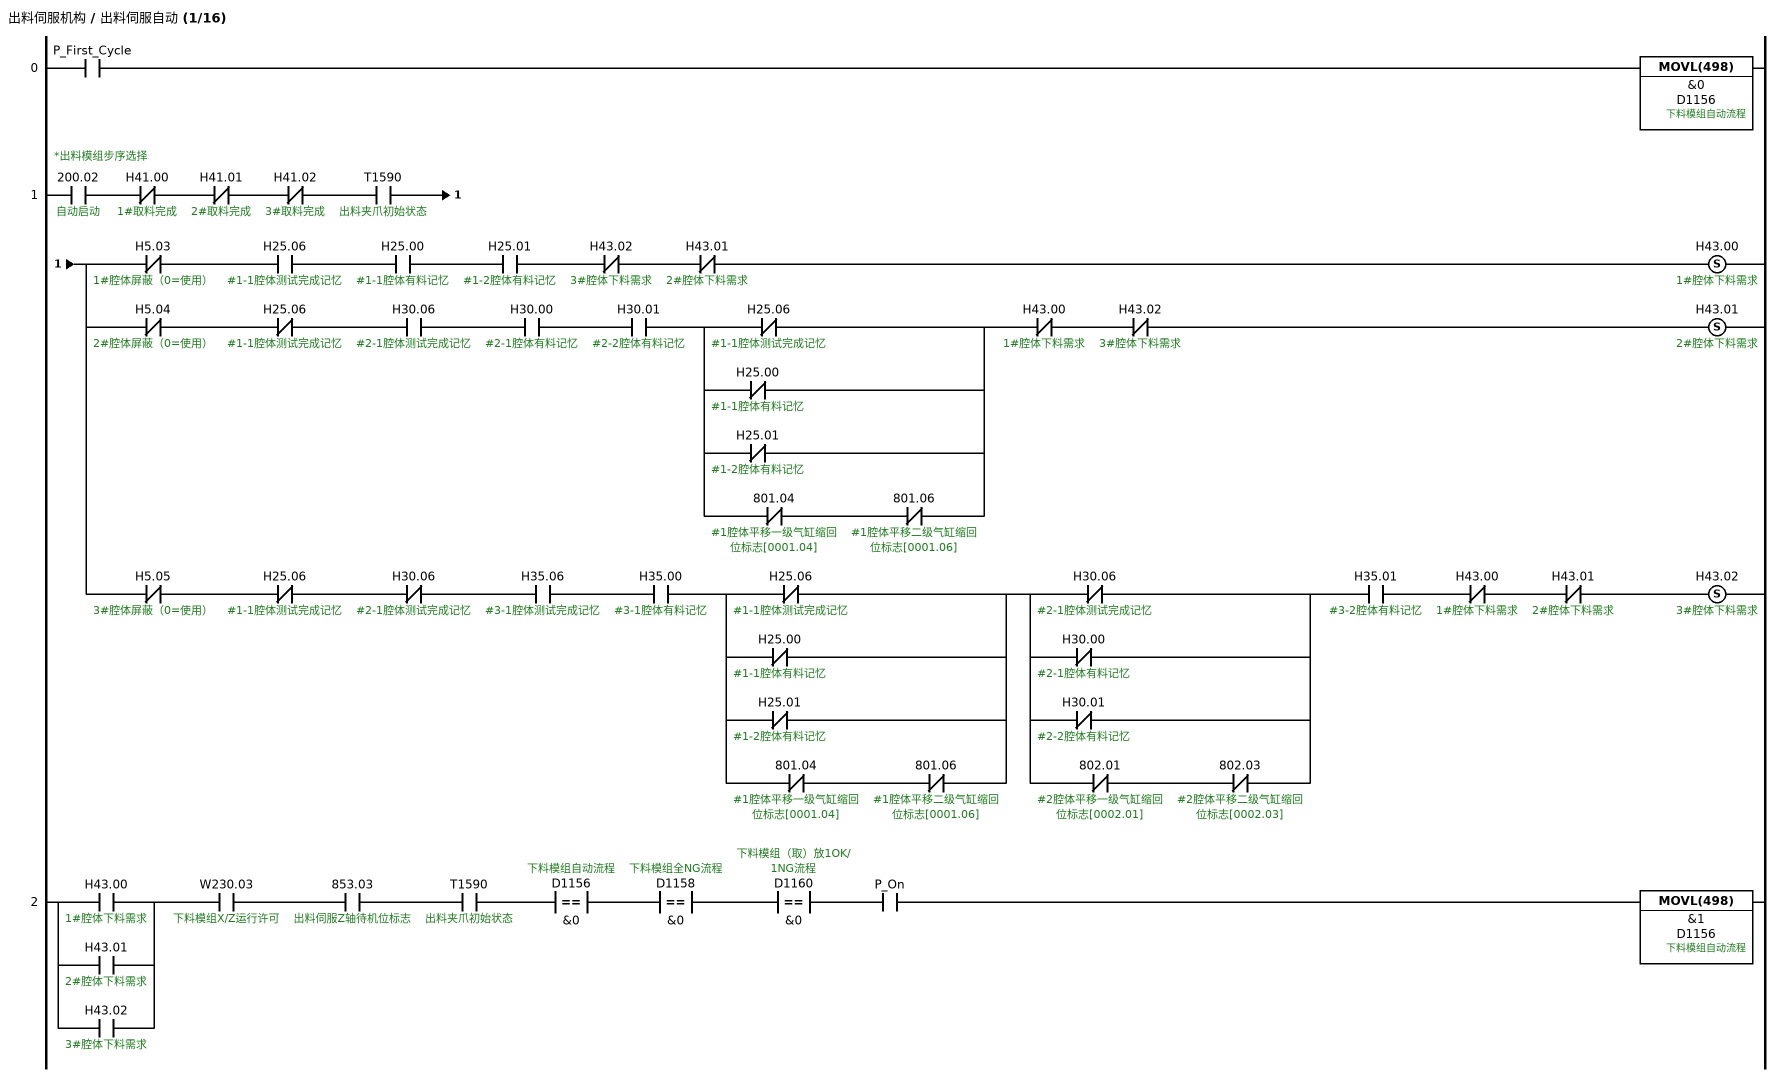
; rung 0
LD P_First_Cycle
MOVL(498) &0 D1156  ; 下料模组自动流程
; rung 1: *出料模组步序选择
LD 200.02  ; 自动启动
ANDNOT H41.00  ; 1#取料完成
ANDNOT H41.01  ; 2#取料完成
ANDNOT H41.02  ; 3#取料完成
AND T1590  ; 出料夹爪初始状态
OUT TR0
ANDNOT H5.03  ; 1#腔体屏蔽（0=使用）
AND H25.06  ; #1-1腔体测试完成记忆
AND H25.00  ; #1-1腔体有料记忆
AND H25.01  ; #1-2腔体有料记忆
ANDNOT H43.02  ; 3#腔体下料需求
ANDNOT H43.01  ; 2#腔体下料需求
SET H43.00  ; 1#腔体下料需求
LD TR0
ANDNOT H5.04  ; 2#腔体屏蔽（0=使用）
ANDNOT H25.06  ; #1-1腔体测试完成记忆
AND H30.06  ; #2-1腔体测试完成记忆
AND H30.00  ; #2-1腔体有料记忆
AND H30.01  ; #2-2腔体有料记忆
LDNOT H25.06  ; #1-1腔体测试完成记忆
ORNOT H25.00  ; #1-1腔体有料记忆
ORNOT H25.01  ; #1-2腔体有料记忆
LDNOT 801.04  ; #1腔体平移一级气缸缩回位标志[0001.04]
ANDNOT 801.06  ; #1腔体平移二级气缸缩回位标志[0001.06]
ORLD
ANDLD
ANDNOT H43.00  ; 1#腔体下料需求
ANDNOT H43.02  ; 3#腔体下料需求
SET H43.01  ; 2#腔体下料需求
LD TR0
ANDNOT H5.05  ; 3#腔体屏蔽（0=使用）
ANDNOT H25.06  ; #1-1腔体测试完成记忆
ANDNOT H30.06  ; #2-1腔体测试完成记忆
AND H35.06  ; #3-1腔体测试完成记忆
AND H35.00  ; #3-1腔体有料记忆
LDNOT H25.06  ; #1-1腔体测试完成记忆
ORNOT H25.00  ; #1-1腔体有料记忆
ORNOT H25.01  ; #1-2腔体有料记忆
LDNOT 801.04  ; #1腔体平移一级气缸缩回位标志[0001.04]
ANDNOT 801.06  ; #1腔体平移二级气缸缩回位标志[0001.06]
ORLD
ANDLD
LDNOT H30.06  ; #2-1腔体测试完成记忆
ORNOT H30.00  ; #2-1腔体有料记忆
ORNOT H30.01  ; #2-2腔体有料记忆
LDNOT 802.01  ; #2腔体平移一级气缸缩回位标志[0002.01]
ANDNOT 802.03  ; #2腔体平移二级气缸缩回位标志[0002.03]
ORLD
ANDLD
AND H35.01  ; #3-2腔体有料记忆
ANDNOT H43.00  ; 1#腔体下料需求
ANDNOT H43.01  ; 2#腔体下料需求
SET H43.02  ; 3#腔体下料需求
; rung 2
LD H43.00  ; 1#腔体下料需求
OR H43.01  ; 2#腔体下料需求
OR H43.02  ; 3#腔体下料需求
AND W230.03  ; 下料模组X/Z运行许可
AND 853.03  ; 出料伺服Z轴待机位标志
AND T1590  ; 出料夹爪初始状态
AND=L(301) D1156 &0  ; 下料模组自动流程
AND=L(301) D1158 &0  ; 下料模组全NG流程
AND=L(301) D1160 &0  ; 下料模组（取）放1OK/1NG流程
AND P_On
MOVL(498) &1 D1156  ; 下料模组自动流程

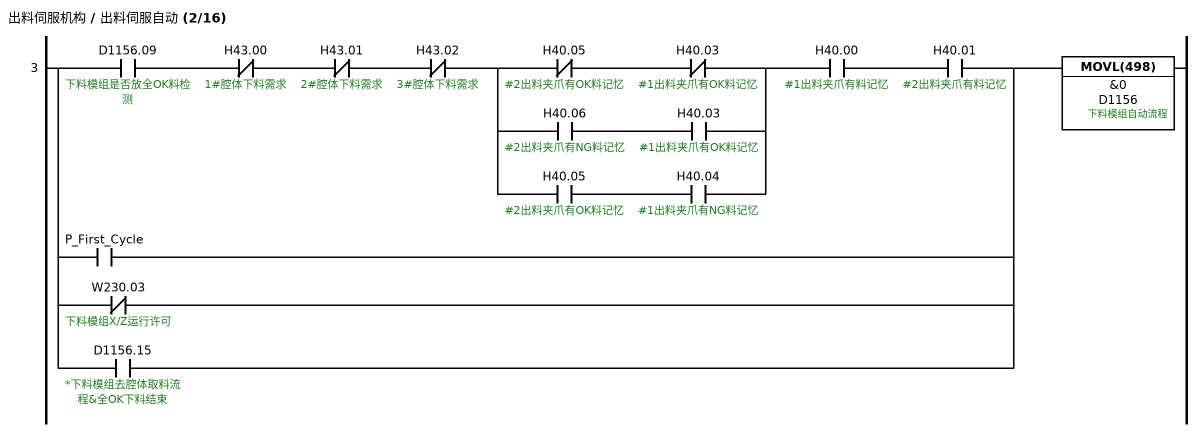
; rung 3
LD D1156.09  ; 下料模组是否放全OK料检测
ANDNOT H43.00  ; 1#腔体下料需求
ANDNOT H43.01  ; 2#腔体下料需求
ANDNOT H43.02  ; 3#腔体下料需求
LDNOT H40.05  ; #2出料夹爪有OK料记忆
ANDNOT H40.03  ; #1出料夹爪有OK料记忆
LD H40.06  ; #2出料夹爪有NG料记忆
AND H40.03  ; #1出料夹爪有OK料记忆
ORLD
LD H40.05  ; #2出料夹爪有OK料记忆
AND H40.04  ; #1出料夹爪有NG料记忆
ORLD
ANDLD
AND H40.00  ; #1出料夹爪有料记忆
AND H40.01  ; #2出料夹爪有料记忆
OR P_First_Cycle
ORNOT W230.03  ; 下料模组X/Z运行许可
OR D1156.15  ; *下料模组去腔体取料流程&全OK下料结束
MOVL(498) &0 D1156  ; 下料模组自动流程

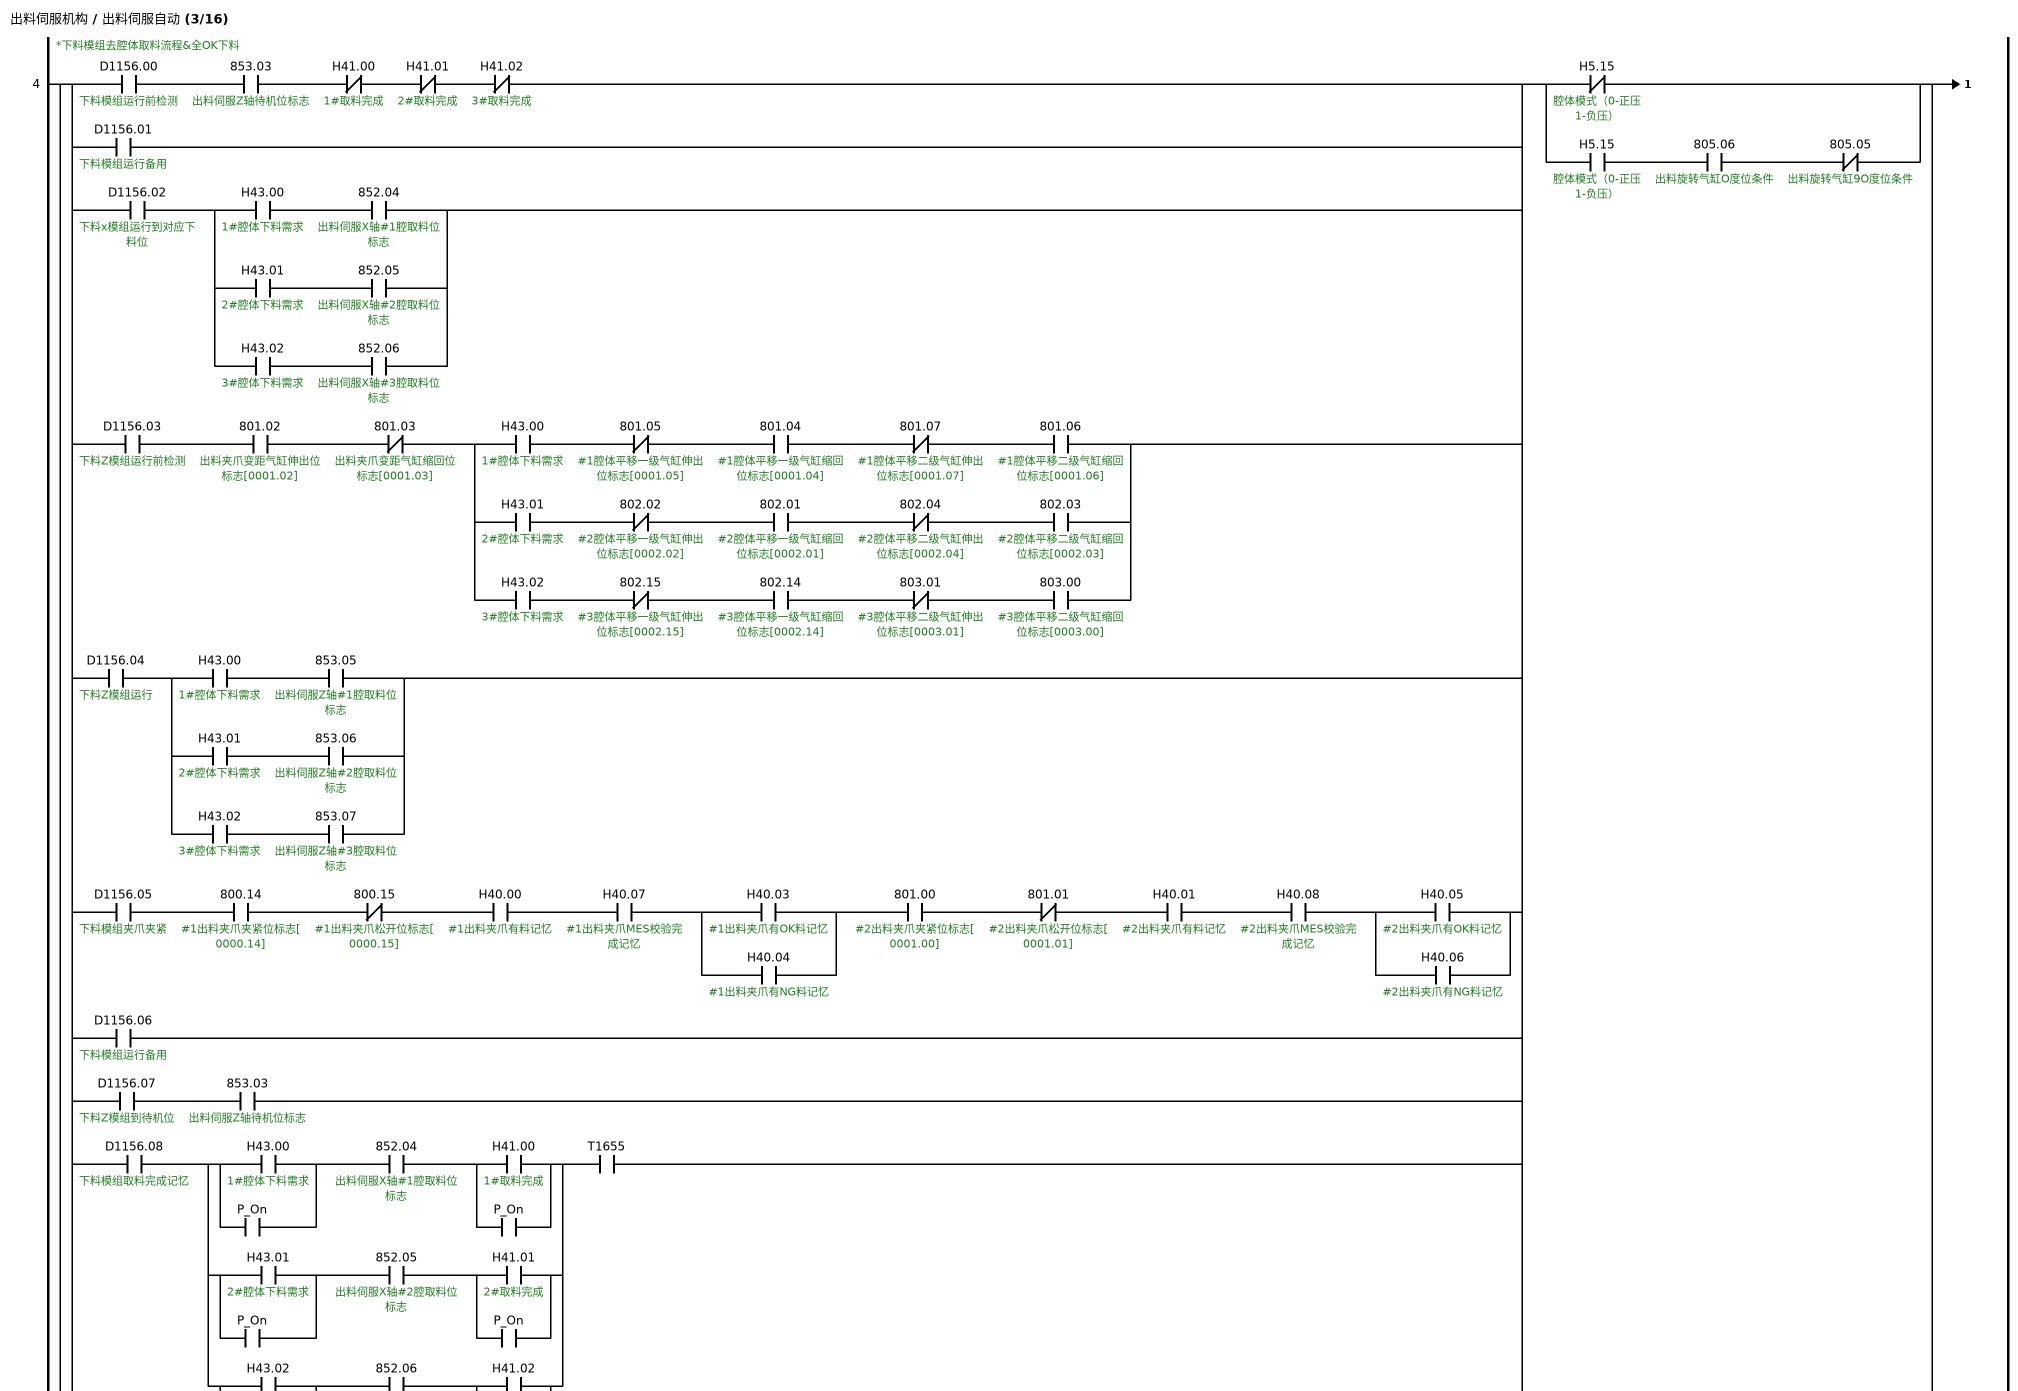

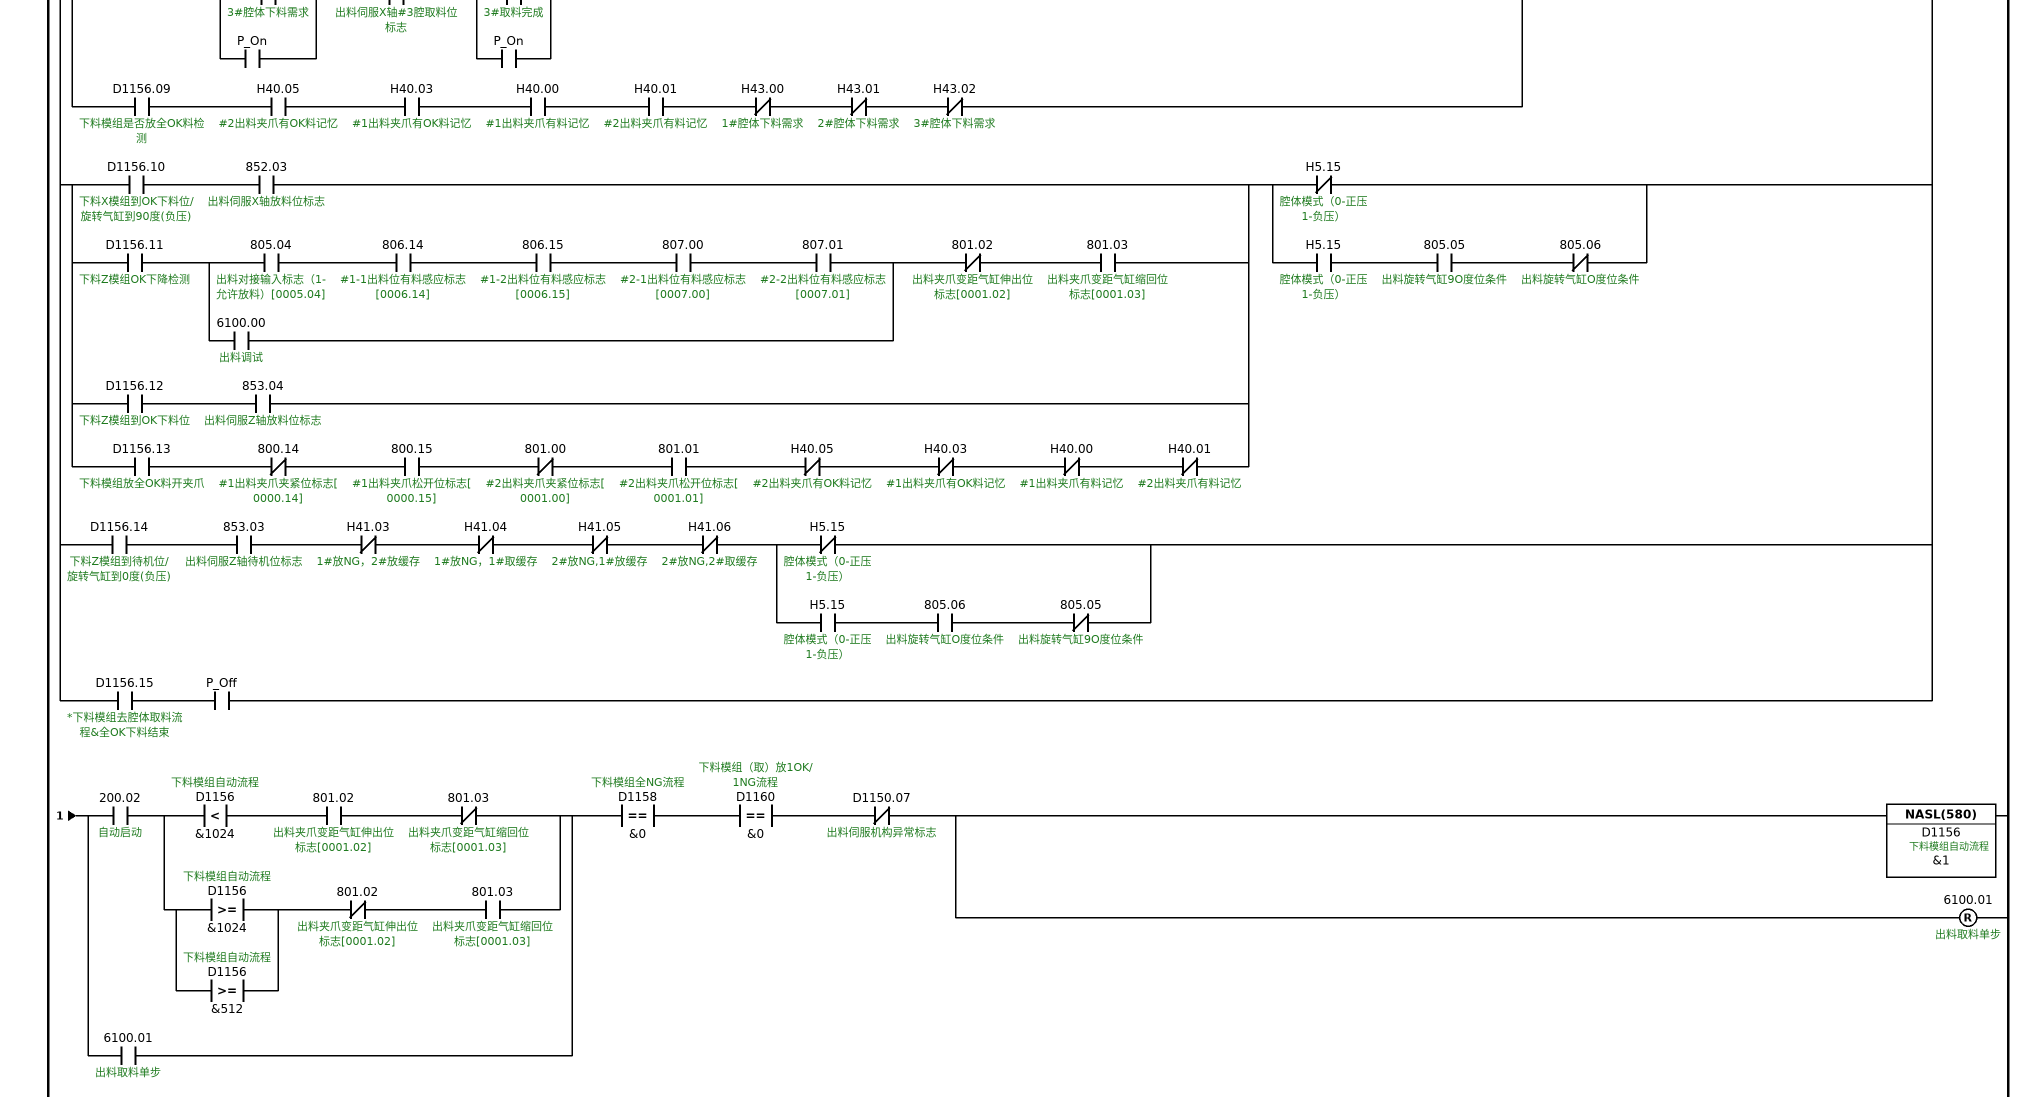
; rung 4: *下料模组去腔体取料流程&全OK下料
LD D1156.00  ; 下料模组运行前检测
AND 853.03  ; 出料伺服Z轴待机位标志
ANDNOT H41.00  ; 1#取料完成
ANDNOT H41.01  ; 2#取料完成
ANDNOT H41.02  ; 3#取料完成
OR D1156.01  ; 下料模组运行备用
LD D1156.02  ; 下料x模组运行到对应下料位
LD H43.00  ; 1#腔体下料需求
AND 852.04  ; 出料伺服X轴#1腔取料位标志
LD H43.01  ; 2#腔体下料需求
AND 852.05  ; 出料伺服X轴#2腔取料位标志
ORLD
LD H43.02  ; 3#腔体下料需求
AND 852.06  ; 出料伺服X轴#3腔取料位标志
ORLD
ANDLD
ORLD
LD D1156.03  ; 下料Z模组运行前检测
AND 801.02  ; 出料夹爪变距气缸伸出位标志[0001.02]
ANDNOT 801.03  ; 出料夹爪变距气缸缩回位标志[0001.03]
LD H43.00  ; 1#腔体下料需求
ANDNOT 801.05  ; #1腔体平移一级气缸伸出位标志[0001.05]
AND 801.04  ; #1腔体平移一级气缸缩回位标志[0001.04]
ANDNOT 801.07  ; #1腔体平移二级气缸伸出位标志[0001.07]
AND 801.06  ; #1腔体平移二级气缸缩回位标志[0001.06]
LD H43.01  ; 2#腔体下料需求
ANDNOT 802.02  ; #2腔体平移一级气缸伸出位标志[0002.02]
AND 802.01  ; #2腔体平移一级气缸缩回位标志[0002.01]
ANDNOT 802.04  ; #2腔体平移二级气缸伸出位标志[0002.04]
AND 802.03  ; #2腔体平移二级气缸缩回位标志[0002.03]
ORLD
LD H43.02  ; 3#腔体下料需求
ANDNOT 802.15  ; #3腔体平移一级气缸伸出位标志[0002.15]
AND 802.14  ; #3腔体平移一级气缸缩回位标志[0002.14]
ANDNOT 803.01  ; #3腔体平移二级气缸伸出位标志[0003.01]
AND 803.00  ; #3腔体平移二级气缸缩回位标志[0003.00]
ORLD
ANDLD
ORLD
LD D1156.04  ; 下料Z模组运行
LD H43.00  ; 1#腔体下料需求
AND 853.05  ; 出料伺服Z轴#1腔取料位标志
LD H43.01  ; 2#腔体下料需求
AND 853.06  ; 出料伺服Z轴#2腔取料位标志
ORLD
LD H43.02  ; 3#腔体下料需求
AND 853.07  ; 出料伺服Z轴#3腔取料位标志
ORLD
ANDLD
ORLD
LD D1156.05  ; 下料模组夹爪夹紧
AND 800.14  ; #1出料夹爪夹紧位标志[0000.14]
ANDNOT 800.15  ; #1出料夹爪松开位标志[0000.15]
AND H40.00  ; #1出料夹爪有料记忆
AND H40.07  ; #1出料夹爪MES校验完成记忆  // 20190115新增
LD H40.03  ; #1出料夹爪有OK料记忆
OR H40.04  ; #1出料夹爪有NG料记忆
ANDLD
AND 801.00  ; #2出料夹爪夹紧位标志[0001.00]
ANDNOT 801.01  ; #2出料夹爪松开位标志[0001.01]
AND H40.01  ; #2出料夹爪有料记忆
AND H40.08  ; #2出料夹爪MES校验完成记忆  // 20190115新增
LD H40.05  ; #2出料夹爪有OK料记忆
OR H40.06  ; #2出料夹爪有NG料记忆
ANDLD
ORLD
OR D1156.06  ; 下料模组运行备用
LD D1156.07  ; 下料Z模组到待机位
AND 853.03  ; 出料伺服Z轴待机位标志
ORLD
LD D1156.08  ; 下料模组取料完成记忆
LD H43.00  ; 1#腔体下料需求
OR P_On
AND 852.04  ; 出料伺服X轴#1腔取料位标志
LD H41.00  ; 1#取料完成
OR P_On
ANDLD
LD H43.01  ; 2#腔体下料需求
OR P_On
AND 852.05  ; 出料伺服X轴#2腔取料位标志
LD H41.01  ; 2#取料完成
OR P_On
ANDLD
ORLD
LD H43.02  ; 3#腔体下料需求
OR P_On
AND 852.06  ; 出料伺服X轴#3腔取料位标志
LD H41.02  ; 3#取料完成
OR P_On
ANDLD
ORLD
ANDLD
AND T1655
ORLD
LD D1156.09  ; 下料模组是否放全OK料检测
AND H40.05  ; #2出料夹爪有OK料记忆
AND H40.03  ; #1出料夹爪有OK料记忆
AND H40.00  ; #1出料夹爪有料记忆
AND H40.01  ; #2出料夹爪有料记忆
ANDNOT H43.00  ; 1#腔体下料需求
ANDNOT H43.01  ; 2#腔体下料需求
ANDNOT H43.02  ; 3#腔体下料需求
ORLD
LDNOT H5.15  ; 腔体模式（0-正压 1-负压）
LD H5.15  ; 腔体模式（0-正压 1-负压）
AND 805.06  ; 出料旋转气缸O度位条件
ANDNOT 805.05  ; 出料旋转气缸9O度位条件
ORLD
ANDLD
LD D1156.10  ; 下料X模组到OK下料位/旋转气缸到90度(负压)
AND 852.03  ; 出料伺服X轴放料位标志
LD D1156.11  ; 下料Z模组OK下降检测
LD 805.04  ; 出料对接输入标志（1-允许放料）[0005.04]
AND 806.14  ; #1-1出料位有料感应标志[0006.14]
AND 806.15  ; #1-2出料位有料感应标志[0006.15]
AND 807.00  ; #2-1出料位有料感应标志[0007.00]
AND 807.01  ; #2-2出料位有料感应标志[0007.01]
OR 6100.00  ; 出料调试
ANDLD
ANDNOT 801.02  ; 出料夹爪变距气缸伸出位标志[0001.02]
AND 801.03  ; 出料夹爪变距气缸缩回位标志[0001.03]
ORLD
LD D1156.12  ; 下料Z模组到OK下料位
AND 853.04  ; 出料伺服Z轴放料位标志
ORLD
LD D1156.13  ; 下料模组放全OK料开夹爪
ANDNOT 800.14  ; #1出料夹爪夹紧位标志[0000.14]
AND 800.15  ; #1出料夹爪松开位标志[0000.15]
ANDNOT 801.00  ; #2出料夹爪夹紧位标志[0001.00]
AND 801.01  ; #2出料夹爪松开位标志[0001.01]
ANDNOT H40.05  ; #2出料夹爪有OK料记忆
ANDNOT H40.03  ; #1出料夹爪有OK料记忆
ANDNOT H40.00  ; #1出料夹爪有料记忆
ANDNOT H40.01  ; #2出料夹爪有料记忆
ORLD
LDNOT H5.15  ; 腔体模式（0-正压 1-负压）
LD H5.15  ; 腔体模式（0-正压 1-负压）
AND 805.05  ; 出料旋转气缸9O度位条件
ANDNOT 805.06  ; 出料旋转气缸O度位条件
ORLD
ANDLD
ORLD
LD D1156.14  ; 下料Z模组到待机位/旋转气缸到0度(负压)
AND 853.03  ; 出料伺服Z轴待机位标志
ANDNOT H41.03  ; 1#放NG，2#放缓存
ANDNOT H41.04  ; 1#放NG，1#取缓存
ANDNOT H41.05  ; 2#放NG,1#放缓存
ANDNOT H41.06  ; 2#放NG,2#取缓存
LDNOT H5.15  ; 腔体模式（0-正压 1-负压）
LD H5.15  ; 腔体模式（0-正压 1-负压）
AND 805.06  ; 出料旋转气缸O度位条件
ANDNOT 805.05  ; 出料旋转气缸9O度位条件
ORLD
ANDLD
ORLD
LD D1156.15  ; *下料模组去腔体取料流程&全OK下料结束
AND P_Off
ORLD
LD 200.02  ; 自动启动
LD<(310) D1156 &1024  ; 下料模组自动流程
AND 801.02  ; 出料夹爪变距气缸伸出位标志[0001.02]
ANDNOT 801.03  ; 出料夹爪变距气缸缩回位标志[0001.03]
LD>=(325) D1156 &1024  ; 下料模组自动流程
OR>=(325) D1156 &512  ; 下料模组自动流程
ANDNOT 801.02  ; 出料夹爪变距气缸伸出位标志[0001.02]
AND 801.03  ; 出料夹爪变距气缸缩回位标志[0001.03]
ORLD
ANDLD
OR 6100.01  ; 出料取料单步
ANDLD
AND=L(301) D1158 &0  ; 下料模组全NG流程
AND=L(301) D1160 &0  ; 下料模组（取）放1OK/1NG流程
ANDNOT D1150.07  ; 出料伺服机构异常标志
NASL(580) D1156 &1  ; 下料模组自动流程
RSET 6100.01  ; 出料取料单步

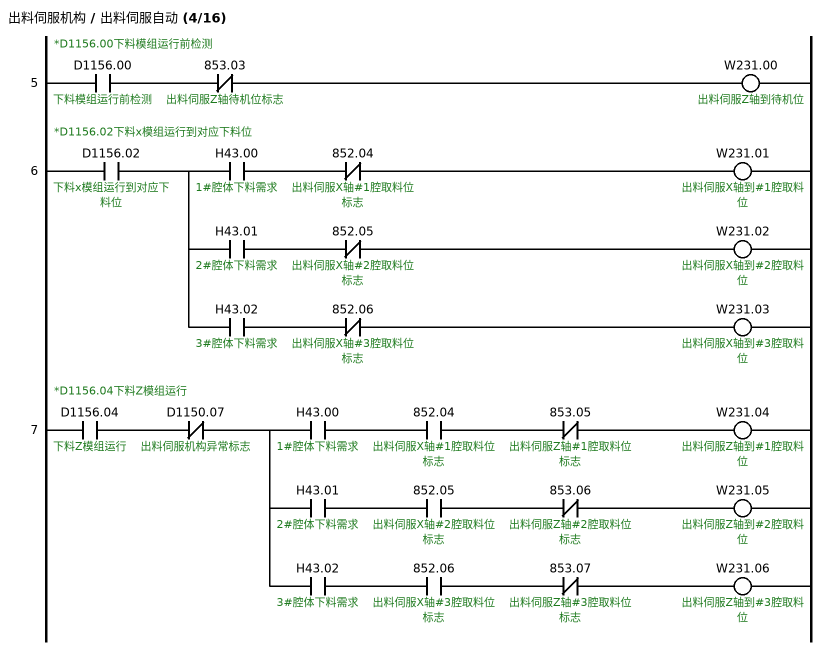
; rung 5: *D1156.00下料模组运行前检测
LD D1156.00  ; 下料模组运行前检测
ANDNOT 853.03  ; 出料伺服Z轴待机位标志
OUT W231.00  ; 出料伺服Z轴到待机位
; rung 6: *D1156.02下料x模组运行到对应下料位
LD D1156.02  ; 下料x模组运行到对应下料位
OUT TR0
AND H43.00  ; 1#腔体下料需求
ANDNOT 852.04  ; 出料伺服X轴#1腔取料位标志
OUT W231.01  ; 出料伺服X轴到#1腔取料位
LD TR0
AND H43.01  ; 2#腔体下料需求
ANDNOT 852.05  ; 出料伺服X轴#2腔取料位标志
OUT W231.02  ; 出料伺服X轴到#2腔取料位
LD TR0
AND H43.02  ; 3#腔体下料需求
ANDNOT 852.06  ; 出料伺服X轴#3腔取料位标志
OUT W231.03  ; 出料伺服X轴到#3腔取料位
; rung 7: *D1156.04下料Z模组运行
LD D1156.04  ; 下料Z模组运行
ANDNOT D1150.07  ; 出料伺服机构异常标志
OUT TR0
AND H43.00  ; 1#腔体下料需求
AND 852.04  ; 出料伺服X轴#1腔取料位标志
ANDNOT 853.05  ; 出料伺服Z轴#1腔取料位标志
OUT W231.04  ; 出料伺服Z轴到#1腔取料位
LD TR0
AND H43.01  ; 2#腔体下料需求
AND 852.05  ; 出料伺服X轴#2腔取料位标志
ANDNOT 853.06  ; 出料伺服Z轴#2腔取料位标志
OUT W231.05  ; 出料伺服Z轴到#2腔取料位
LD TR0
AND H43.02  ; 3#腔体下料需求
AND 852.06  ; 出料伺服X轴#3腔取料位标志
ANDNOT 853.07  ; 出料伺服Z轴#3腔取料位标志
OUT W231.06  ; 出料伺服Z轴到#3腔取料位

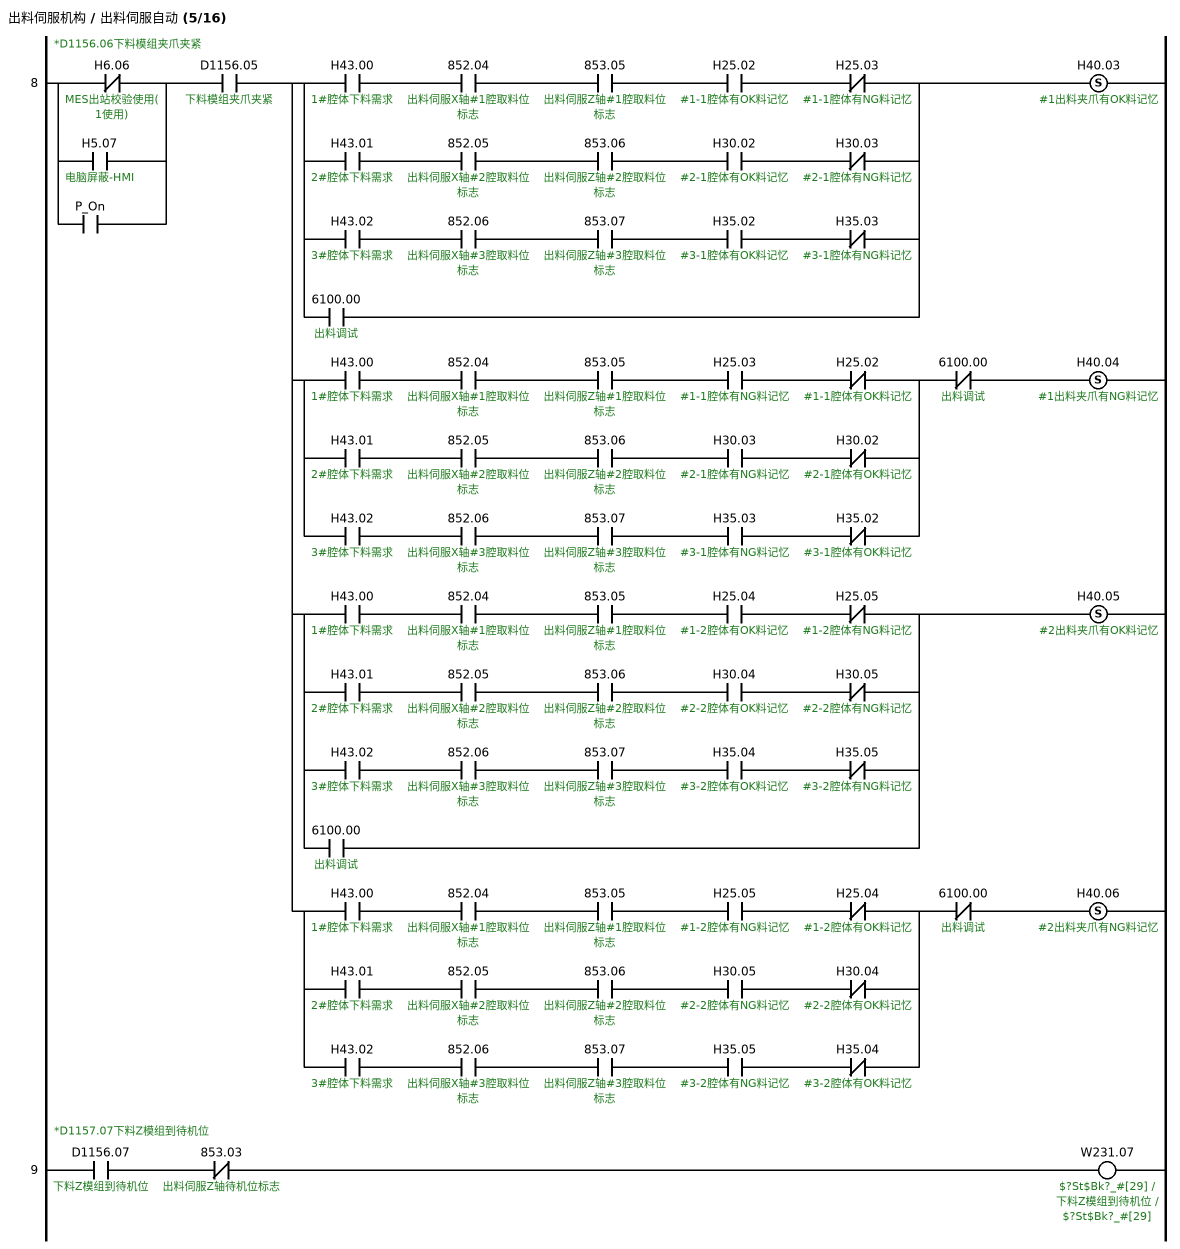
; rung 8: *D1156.06下料模组夹爪夹紧
LDNOT H6.06  ; MES出站校验使用(1使用)
OR H5.07  ; 电脑屏蔽-HMI
OR P_On
AND D1156.05  ; 下料模组夹爪夹紧
OUT TR0
LD H43.00  ; 1#腔体下料需求
AND 852.04  ; 出料伺服X轴#1腔取料位标志
AND 853.05  ; 出料伺服Z轴#1腔取料位标志
AND H25.02  ; #1-1腔体有OK料记忆
ANDNOT H25.03  ; #1-1腔体有NG料记忆
LD H43.01  ; 2#腔体下料需求
AND 852.05  ; 出料伺服X轴#2腔取料位标志
AND 853.06  ; 出料伺服Z轴#2腔取料位标志
AND H30.02  ; #2-1腔体有OK料记忆
ANDNOT H30.03  ; #2-1腔体有NG料记忆
ORLD
LD H43.02  ; 3#腔体下料需求
AND 852.06  ; 出料伺服X轴#3腔取料位标志
AND 853.07  ; 出料伺服Z轴#3腔取料位标志
AND H35.02  ; #3-1腔体有OK料记忆
ANDNOT H35.03  ; #3-1腔体有NG料记忆
ORLD
OR 6100.00  ; 出料调试
ANDLD
SET H40.03  ; #1出料夹爪有OK料记忆
LD TR0
LD H43.00  ; 1#腔体下料需求
AND 852.04  ; 出料伺服X轴#1腔取料位标志
AND 853.05  ; 出料伺服Z轴#1腔取料位标志
AND H25.03  ; #1-1腔体有NG料记忆
ANDNOT H25.02  ; #1-1腔体有OK料记忆
LD H43.01  ; 2#腔体下料需求
AND 852.05  ; 出料伺服X轴#2腔取料位标志
AND 853.06  ; 出料伺服Z轴#2腔取料位标志
AND H30.03  ; #2-1腔体有NG料记忆
ANDNOT H30.02  ; #2-1腔体有OK料记忆
ORLD
LD H43.02  ; 3#腔体下料需求
AND 852.06  ; 出料伺服X轴#3腔取料位标志
AND 853.07  ; 出料伺服Z轴#3腔取料位标志
AND H35.03  ; #3-1腔体有NG料记忆
ANDNOT H35.02  ; #3-1腔体有OK料记忆
ORLD
ANDLD
ANDNOT 6100.00  ; 出料调试
SET H40.04  ; #1出料夹爪有NG料记忆
LD TR0
LD H43.00  ; 1#腔体下料需求
AND 852.04  ; 出料伺服X轴#1腔取料位标志
AND 853.05  ; 出料伺服Z轴#1腔取料位标志
AND H25.04  ; #1-2腔体有OK料记忆
ANDNOT H25.05  ; #1-2腔体有NG料记忆
LD H43.01  ; 2#腔体下料需求
AND 852.05  ; 出料伺服X轴#2腔取料位标志
AND 853.06  ; 出料伺服Z轴#2腔取料位标志
AND H30.04  ; #2-2腔体有OK料记忆
ANDNOT H30.05  ; #2-2腔体有NG料记忆
ORLD
LD H43.02  ; 3#腔体下料需求
AND 852.06  ; 出料伺服X轴#3腔取料位标志
AND 853.07  ; 出料伺服Z轴#3腔取料位标志
AND H35.04  ; #3-2腔体有OK料记忆
ANDNOT H35.05  ; #3-2腔体有NG料记忆
ORLD
OR 6100.00  ; 出料调试
ANDLD
SET H40.05  ; #2出料夹爪有OK料记忆
LD TR0
LD H43.00  ; 1#腔体下料需求
AND 852.04  ; 出料伺服X轴#1腔取料位标志
AND 853.05  ; 出料伺服Z轴#1腔取料位标志
AND H25.05  ; #1-2腔体有NG料记忆
ANDNOT H25.04  ; #1-2腔体有OK料记忆
LD H43.01  ; 2#腔体下料需求
AND 852.05  ; 出料伺服X轴#2腔取料位标志
AND 853.06  ; 出料伺服Z轴#2腔取料位标志
AND H30.05  ; #2-2腔体有NG料记忆
ANDNOT H30.04  ; #2-2腔体有OK料记忆
ORLD
LD H43.02  ; 3#腔体下料需求
AND 852.06  ; 出料伺服X轴#3腔取料位标志
AND 853.07  ; 出料伺服Z轴#3腔取料位标志
AND H35.05  ; #3-2腔体有NG料记忆
ANDNOT H35.04  ; #3-2腔体有OK料记忆
ORLD
ANDLD
ANDNOT 6100.00  ; 出料调试
SET H40.06  ; #2出料夹爪有NG料记忆
; rung 9: *D1157.07下料Z模组到待机位
LD D1156.07  ; 下料Z模组到待机位
ANDNOT 853.03  ; 出料伺服Z轴待机位标志
OUT W231.07  ; $?St$Bk?_#[29] / 下料Z模组到待机位 / $?St$Bk?_#[29]

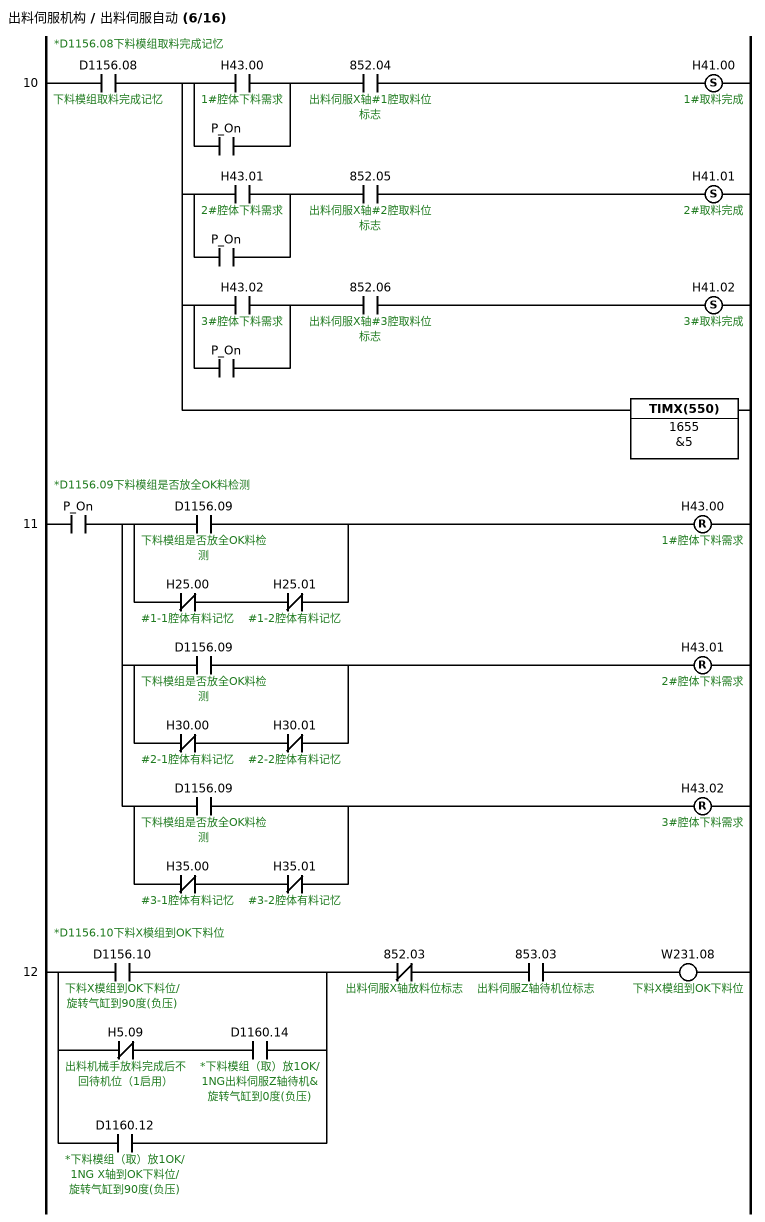
; rung 10: *D1156.08下料模组取料完成记忆
LD D1156.08  ; 下料模组取料完成记忆
OUT TR0
LD H43.00  ; 1#腔体下料需求
OR P_On
ANDLD
AND 852.04  ; 出料伺服X轴#1腔取料位标志
SET H41.00  ; 1#取料完成
LD TR0
LD H43.01  ; 2#腔体下料需求
OR P_On
ANDLD
AND 852.05  ; 出料伺服X轴#2腔取料位标志
SET H41.01  ; 2#取料完成
LD TR0
LD H43.02  ; 3#腔体下料需求
OR P_On
ANDLD
AND 852.06  ; 出料伺服X轴#3腔取料位标志
SET H41.02  ; 3#取料完成
LD TR0
TIMX(550) 1655 &5
; rung 11: *D1156.09下料模组是否放全OK料检测
LD P_On
OUT TR0
LD D1156.09  ; 下料模组是否放全OK料检测
LDNOT H25.00  ; #1-1腔体有料记忆
ANDNOT H25.01  ; #1-2腔体有料记忆
ORLD
ANDLD
RSET H43.00  ; 1#腔体下料需求
LD TR0
LD D1156.09  ; 下料模组是否放全OK料检测
LDNOT H30.00  ; #2-1腔体有料记忆
ANDNOT H30.01  ; #2-2腔体有料记忆
ORLD
ANDLD
RSET H43.01  ; 2#腔体下料需求
LD TR0
LD D1156.09  ; 下料模组是否放全OK料检测
LDNOT H35.00  ; #3-1腔体有料记忆
ANDNOT H35.01  ; #3-2腔体有料记忆
ORLD
ANDLD
RSET H43.02  ; 3#腔体下料需求
; rung 12: *D1156.10下料X模组到OK下料位
LD D1156.10  ; 下料X模组到OK下料位/旋转气缸到90度(负压)
LDNOT H5.09  ; 出料机械手放料完成后不回待机位（1启用）
AND D1160.14  ; *下料模组（取）放1OK/1NG出料伺服Z轴待机&旋转气缸到0度(负压)
ORLD
OR D1160.12  ; *下料模组（取）放1OK/1NG X轴到OK下料位/旋转气缸到90度(负压)
ANDNOT 852.03  ; 出料伺服X轴放料位标志
AND 853.03  ; 出料伺服Z轴待机位标志
OUT W231.08  ; 下料X模组到OK下料位

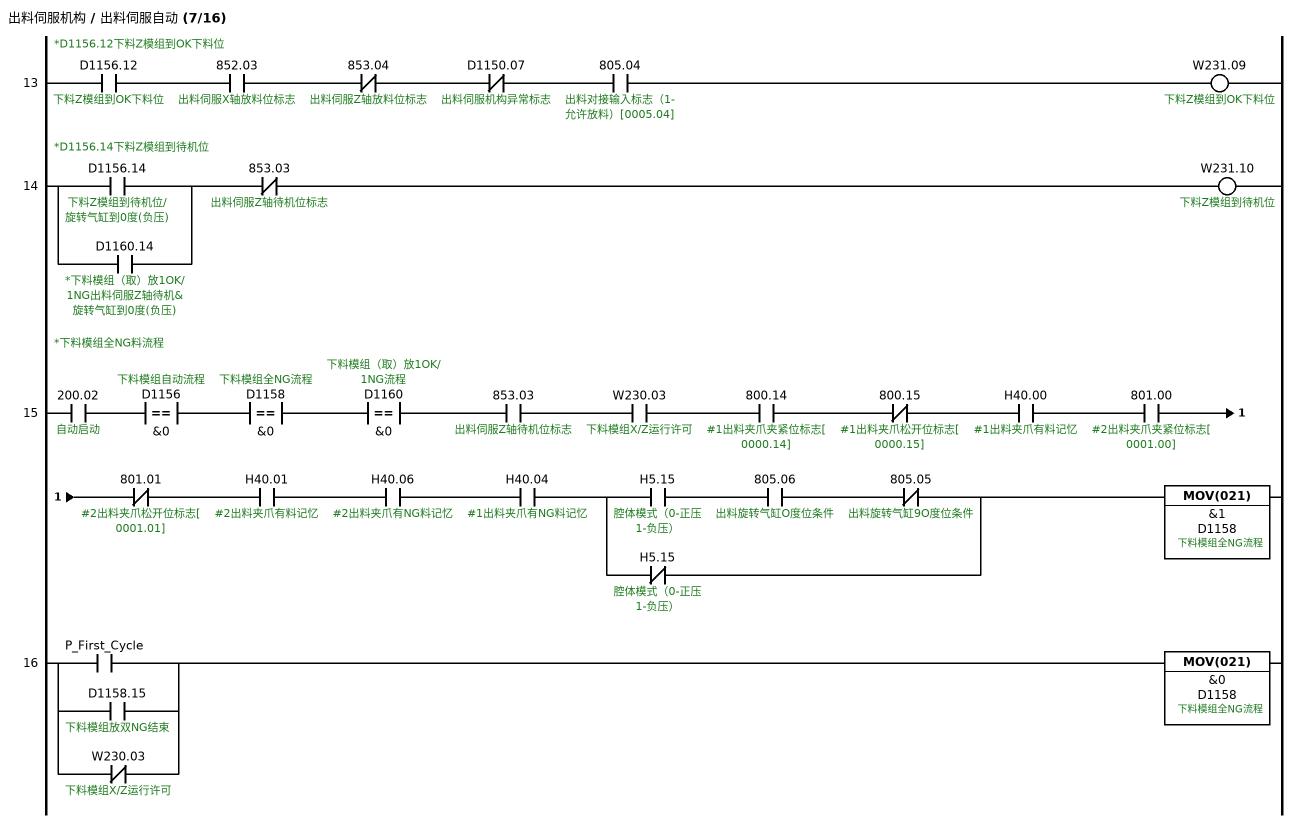
; rung 13: *D1156.12下料Z模组到OK下料位
LD D1156.12  ; 下料Z模组到OK下料位
AND 852.03  ; 出料伺服X轴放料位标志
ANDNOT 853.04  ; 出料伺服Z轴放料位标志
ANDNOT D1150.07  ; 出料伺服机构异常标志
AND 805.04  ; 出料对接输入标志（1-允许放料）[0005.04]
OUT W231.09  ; 下料Z模组到OK下料位
; rung 14: *D1156.14下料Z模组到待机位
LD D1156.14  ; 下料Z模组到待机位/旋转气缸到0度(负压)
OR D1160.14  ; *下料模组（取）放1OK/1NG出料伺服Z轴待机&旋转气缸到0度(负压)
ANDNOT 853.03  ; 出料伺服Z轴待机位标志
OUT W231.10  ; 下料Z模组到待机位
; rung 15: *下料模组全NG料流程
LD 200.02  ; 自动启动
AND=L(301) D1156 &0  ; 下料模组自动流程
AND=L(301) D1158 &0  ; 下料模组全NG流程
AND=L(301) D1160 &0  ; 下料模组（取）放1OK/1NG流程
AND 853.03  ; 出料伺服Z轴待机位标志
AND W230.03  ; 下料模组X/Z运行许可
AND 800.14  ; #1出料夹爪夹紧位标志[0000.14]
ANDNOT 800.15  ; #1出料夹爪松开位标志[0000.15]
AND H40.00  ; #1出料夹爪有料记忆
AND 801.00  ; #2出料夹爪夹紧位标志[0001.00]
ANDNOT 801.01  ; #2出料夹爪松开位标志[0001.01]
AND H40.01  ; #2出料夹爪有料记忆
AND H40.06  ; #2出料夹爪有NG料记忆
AND H40.04  ; #1出料夹爪有NG料记忆
LD H5.15  ; 腔体模式（0-正压 1-负压）
AND 805.06  ; 出料旋转气缸O度位条件
ANDNOT 805.05  ; 出料旋转气缸9O度位条件
ORNOT H5.15  ; 腔体模式（0-正压 1-负压）
ANDLD
MOV(021) &1 D1158  ; 下料模组全NG流程
; rung 16
LD P_First_Cycle
OR D1158.15  ; 下料模组放双NG结束
ORNOT W230.03  ; 下料模组X/Z运行许可
MOV(021) &0 D1158  ; 下料模组全NG流程

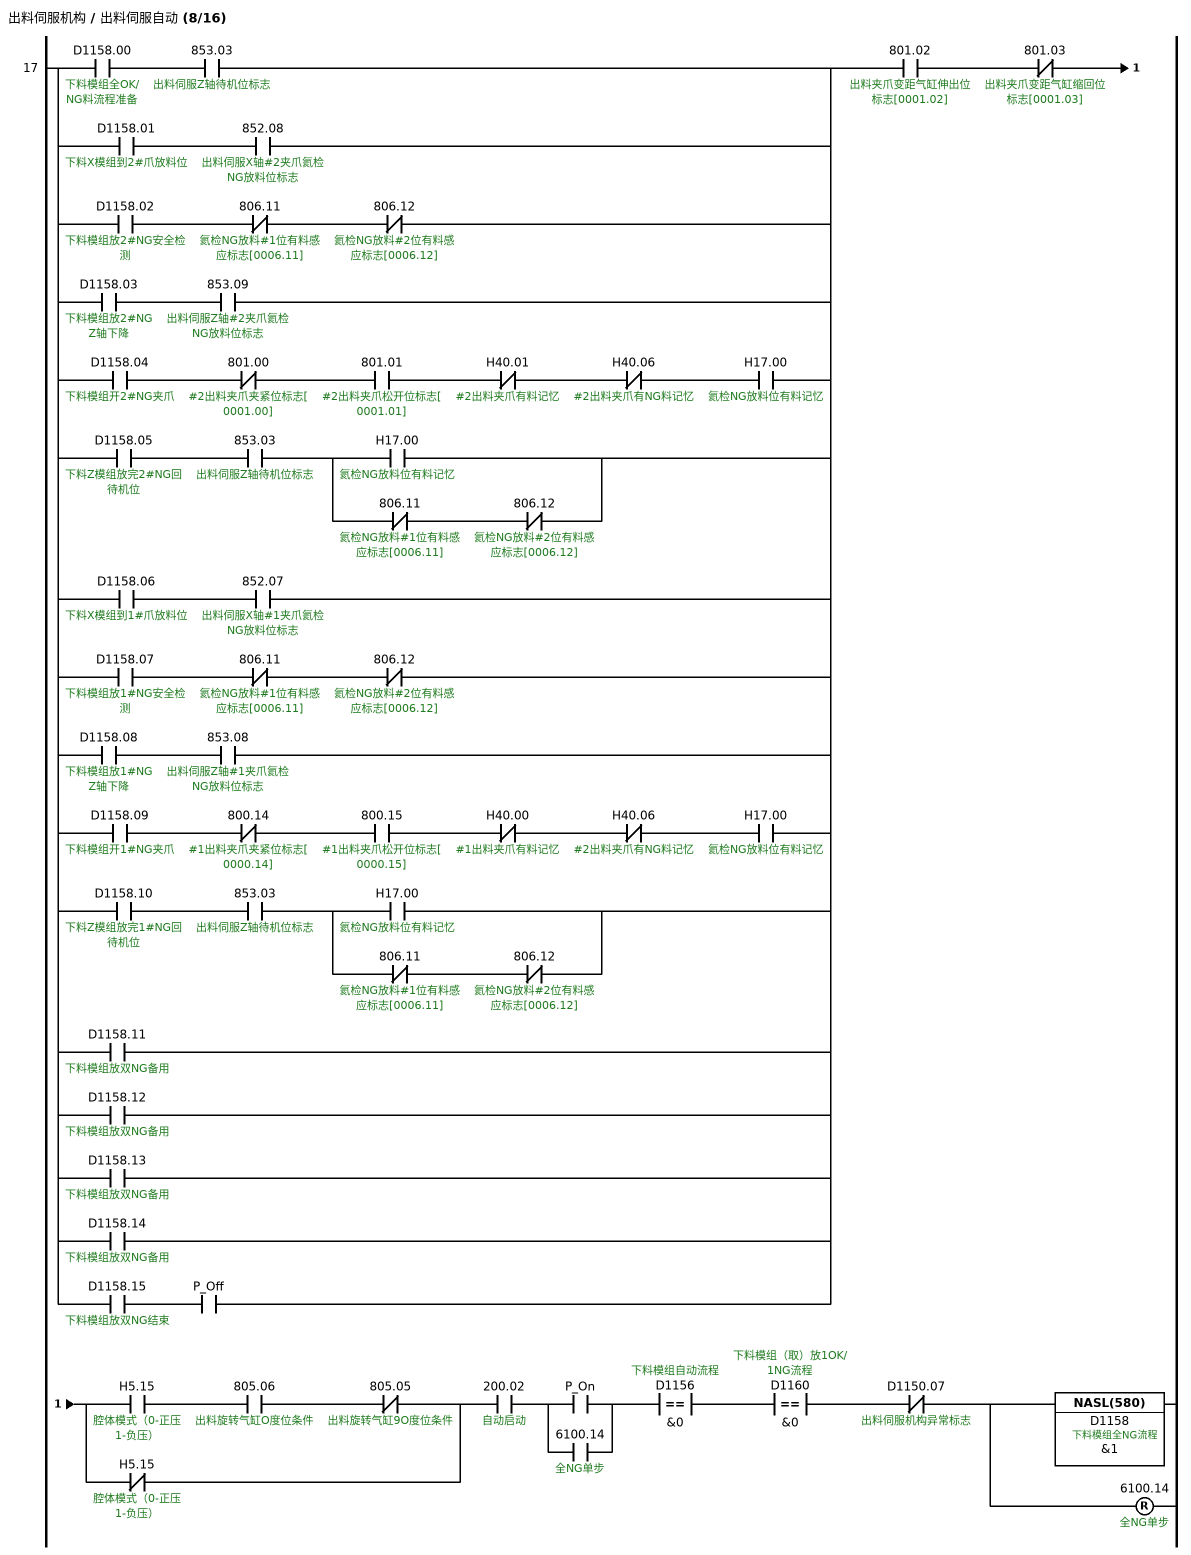
; rung 17
LD D1158.00  ; 下料模组全OK/NG料流程准备
AND 853.03  ; 出料伺服Z轴待机位标志
LD D1158.01  ; 下料X模组到2#爪放料位
AND 852.08  ; 出料伺服X轴#2夹爪氦检NG放料位标志
ORLD
LD D1158.02  ; 下料模组放2#NG安全检测
ANDNOT 806.11  ; 氦检NG放料#1位有料感应标志[0006.11]
ANDNOT 806.12  ; 氦检NG放料#2位有料感应标志[0006.12]
ORLD
LD D1158.03  ; 下料模组放2#NG Z轴下降
AND 853.09  ; 出料伺服Z轴#2夹爪氦检NG放料位标志
ORLD
LD D1158.04  ; 下料模组开2#NG夹爪
ANDNOT 801.00  ; #2出料夹爪夹紧位标志[0001.00]
AND 801.01  ; #2出料夹爪松开位标志[0001.01]
ANDNOT H40.01  ; #2出料夹爪有料记忆
ANDNOT H40.06  ; #2出料夹爪有NG料记忆
AND H17.00  ; 氦检NG放料位有料记忆
ORLD
LD D1158.05  ; 下料Z模组放完2#NG回待机位
AND 853.03  ; 出料伺服Z轴待机位标志
LD H17.00  ; 氦检NG放料位有料记忆
LDNOT 806.11  ; 氦检NG放料#1位有料感应标志[0006.11]
ANDNOT 806.12  ; 氦检NG放料#2位有料感应标志[0006.12]
ORLD
ANDLD
ORLD
LD D1158.06  ; 下料X模组到1#爪放料位
AND 852.07  ; 出料伺服X轴#1夹爪氦检NG放料位标志
ORLD
LD D1158.07  ; 下料模组放1#NG安全检测
ANDNOT 806.11  ; 氦检NG放料#1位有料感应标志[0006.11]
ANDNOT 806.12  ; 氦检NG放料#2位有料感应标志[0006.12]
ORLD
LD D1158.08  ; 下料模组放1#NG Z轴下降
AND 853.08  ; 出料伺服Z轴#1夹爪氦检NG放料位标志
ORLD
LD D1158.09  ; 下料模组开1#NG夹爪
ANDNOT 800.14  ; #1出料夹爪夹紧位标志[0000.14]
AND 800.15  ; #1出料夹爪松开位标志[0000.15]
ANDNOT H40.00  ; #1出料夹爪有料记忆
ANDNOT H40.06  ; #2出料夹爪有NG料记忆
AND H17.00  ; 氦检NG放料位有料记忆
ORLD
LD D1158.10  ; 下料Z模组放完1#NG回待机位
AND 853.03  ; 出料伺服Z轴待机位标志
LD H17.00  ; 氦检NG放料位有料记忆
LDNOT 806.11  ; 氦检NG放料#1位有料感应标志[0006.11]
ANDNOT 806.12  ; 氦检NG放料#2位有料感应标志[0006.12]
ORLD
ANDLD
ORLD
OR D1158.11  ; 下料模组放双NG备用
OR D1158.12  ; 下料模组放双NG备用
OR D1158.13  ; 下料模组放双NG备用
OR D1158.14  ; 下料模组放双NG备用
LD D1158.15  ; 下料模组放双NG结束
AND P_Off
ORLD
AND 801.02  ; 出料夹爪变距气缸伸出位标志[0001.02]
ANDNOT 801.03  ; 出料夹爪变距气缸缩回位标志[0001.03]
LD H5.15  ; 腔体模式（0-正压 1-负压）
AND 805.06  ; 出料旋转气缸O度位条件
ANDNOT 805.05  ; 出料旋转气缸9O度位条件
ORNOT H5.15  ; 腔体模式（0-正压 1-负压）
ANDLD
AND 200.02  ; 自动启动
LD P_On
OR 6100.14  ; 全NG单步
ANDLD
AND=L(301) D1156 &0  ; 下料模组自动流程
AND=L(301) D1160 &0  ; 下料模组（取）放1OK/1NG流程
ANDNOT D1150.07  ; 出料伺服机构异常标志
NASL(580) D1158 &1  ; 下料模组全NG流程
RSET 6100.14  ; 全NG单步

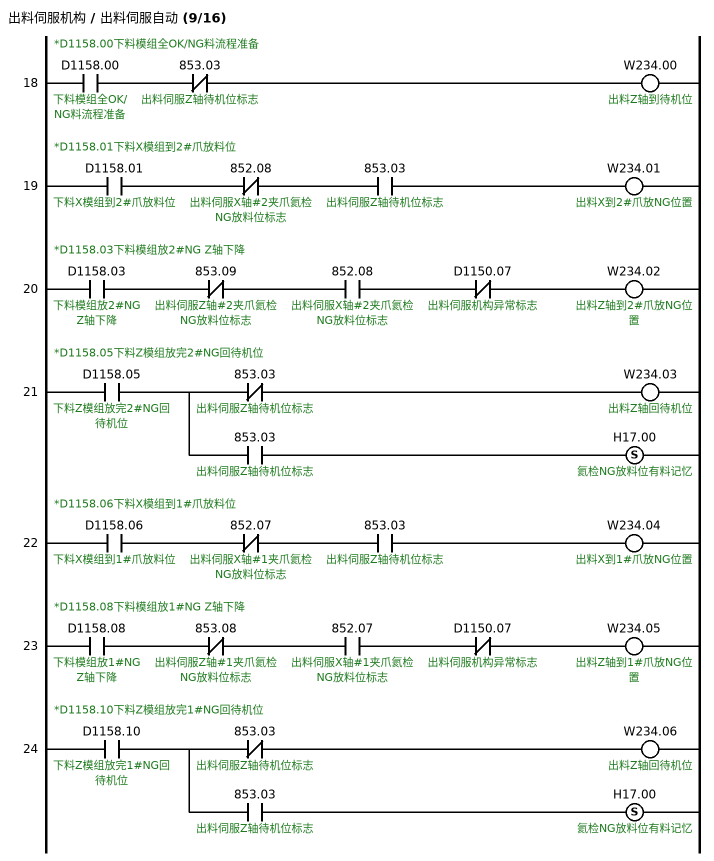
; rung 18: *D1158.00下料模组全OK/NG料流程准备
LD D1158.00  ; 下料模组全OK/NG料流程准备
ANDNOT 853.03  ; 出料伺服Z轴待机位标志
OUT W234.00  ; 出料Z轴到待机位
; rung 19: *D1158.01下料X模组到2#爪放料位
LD D1158.01  ; 下料X模组到2#爪放料位
ANDNOT 852.08  ; 出料伺服X轴#2夹爪氦检NG放料位标志
AND 853.03  ; 出料伺服Z轴待机位标志
OUT W234.01  ; 出料X到2#爪放NG位置
; rung 20: *D1158.03下料模组放2#NG Z轴下降
LD D1158.03  ; 下料模组放2#NG Z轴下降
ANDNOT 853.09  ; 出料伺服Z轴#2夹爪氦检NG放料位标志
AND 852.08  ; 出料伺服X轴#2夹爪氦检NG放料位标志
ANDNOT D1150.07  ; 出料伺服机构异常标志
OUT W234.02  ; 出料Z轴到2#爪放NG位置
; rung 21: *D1158.05下料Z模组放完2#NG回待机位
LD D1158.05  ; 下料Z模组放完2#NG回待机位
OUT TR0
ANDNOT 853.03  ; 出料伺服Z轴待机位标志
OUT W234.03  ; 出料Z轴回待机位
LD TR0
AND 853.03  ; 出料伺服Z轴待机位标志
SET H17.00  ; 氦检NG放料位有料记忆
; rung 22: *D1158.06下料X模组到1#爪放料位
LD D1158.06  ; 下料X模组到1#爪放料位
ANDNOT 852.07  ; 出料伺服X轴#1夹爪氦检NG放料位标志
AND 853.03  ; 出料伺服Z轴待机位标志
OUT W234.04  ; 出料X到1#爪放NG位置
; rung 23: *D1158.08下料模组放1#NG Z轴下降
LD D1158.08  ; 下料模组放1#NG Z轴下降
ANDNOT 853.08  ; 出料伺服Z轴#1夹爪氦检NG放料位标志
AND 852.07  ; 出料伺服X轴#1夹爪氦检NG放料位标志
ANDNOT D1150.07  ; 出料伺服机构异常标志
OUT W234.05  ; 出料Z轴到1#爪放NG位置
; rung 24: *D1158.10下料Z模组放完1#NG回待机位
LD D1158.10  ; 下料Z模组放完1#NG回待机位
OUT TR0
ANDNOT 853.03  ; 出料伺服Z轴待机位标志
OUT W234.06  ; 出料Z轴回待机位
LD TR0
AND 853.03  ; 出料伺服Z轴待机位标志
SET H17.00  ; 氦检NG放料位有料记忆

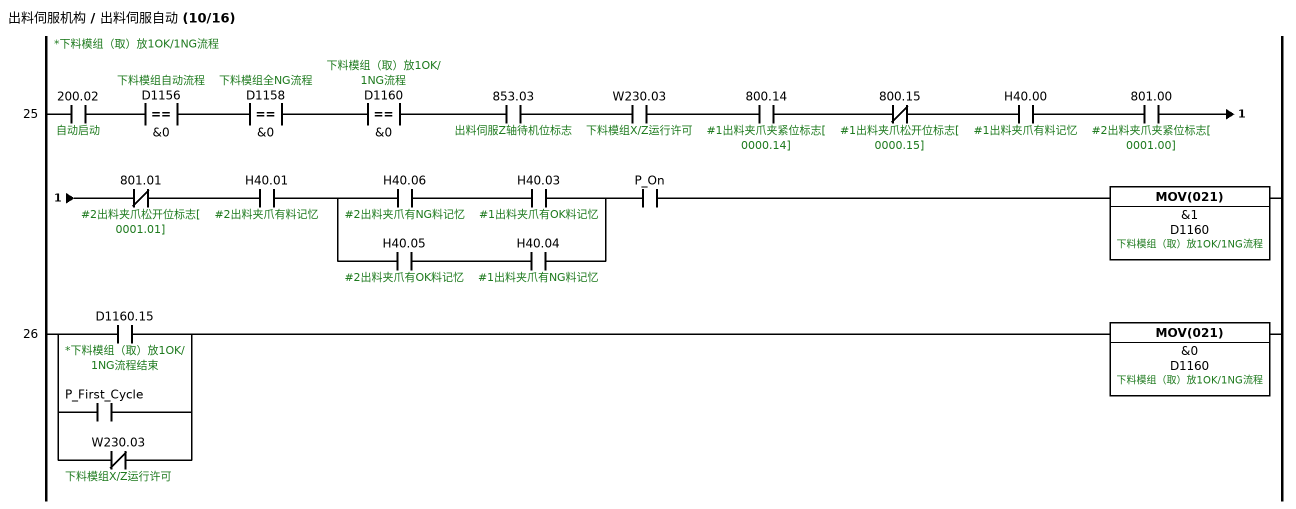
; rung 25: *下料模组（取）放1OK/1NG流程
LD 200.02  ; 自动启动
AND=L(301) D1156 &0  ; 下料模组自动流程
AND=L(301) D1158 &0  ; 下料模组全NG流程
AND=L(301) D1160 &0  ; 下料模组（取）放1OK/1NG流程
AND 853.03  ; 出料伺服Z轴待机位标志
AND W230.03  ; 下料模组X/Z运行许可
AND 800.14  ; #1出料夹爪夹紧位标志[0000.14]
ANDNOT 800.15  ; #1出料夹爪松开位标志[0000.15]
AND H40.00  ; #1出料夹爪有料记忆
AND 801.00  ; #2出料夹爪夹紧位标志[0001.00]
ANDNOT 801.01  ; #2出料夹爪松开位标志[0001.01]
AND H40.01  ; #2出料夹爪有料记忆
LD H40.06  ; #2出料夹爪有NG料记忆
AND H40.03  ; #1出料夹爪有OK料记忆
LD H40.05  ; #2出料夹爪有OK料记忆
AND H40.04  ; #1出料夹爪有NG料记忆
ORLD
ANDLD
AND P_On
MOV(021) &1 D1160  ; 下料模组（取）放1OK/1NG流程
; rung 26
LD D1160.15  ; *下料模组（取）放1OK/1NG流程结束
OR P_First_Cycle
ORNOT W230.03  ; 下料模组X/Z运行许可
MOV(021) &0 D1160  ; 下料模组（取）放1OK/1NG流程

